// TwinCAT 3 PLC project Testing
// ProgramVersion: 3.1.4026.17
// libraries:
//   Tc2_Standard, * (Beckhoff Automation GmbH)
//   Tc2_System, * (Beckhoff Automation GmbH)
//   [TcForge], * (Home)
//   TcUnit, * (www.tcunit.org)
// project tree:
//   POUs/ MAIN.TcPOU, FB_DeviceBase_Probe.TcPOU, FB_DigitalInput_Probe.TcPOU, FB_TwoPosActuator_Probe.TcPOU, FB_AnalogInput_Probe.TcPOU, FB_AnalogOutput_Probe.TcPOU, FB_StateMachine_Probe.TcPOU
//   / Testing.TcTTO
//   Tests/ FB_F_ValidateRequester_Test.TcPOU, FB_BitMatrix64_Test.TcPOU, FB_Permissives_Test.TcPOU, FB_Interlock_Test.TcPOU, FB_AlarmSimple_Test.TcPOU, FB_AlarmLimit_Test.TcPOU, FB_DeviceBase_Test.TcPOU, FB_LPF_FirstOrder_IIR_Test.TcPOU, FB_DigitalOutput_Test.TcPOU, FB_DigitalInput_Test.TcPOU, FB_TwoPosActuator_Test.TcPOU, FB_AnalogInput_Test.TcPOU, FB_AnalogOutput_Test.TcPOU, FB_AlarmThreshold_Test.TcPOU, FB_AlarmDeviation_Test.TcPOU, FB_Step_Test.TcPOU, FB_StateMachine_Test.TcPOU
// (motion and I/O tree: see PLC project tcforge)
// real-time tasks:
//   TASK Testing: cycle T#10ms, priority 2, ADS port 351
//   TASK PlcTask: cycle T#10ms, priority 1, ADS port 350

CONFIGURATION Testing
    RESOURCE PLC ON TwinCAT3
        TASK Testing(INTERVAL := T#10ms, PRIORITY := 2);
        PROGRAM MAIN WITH Testing : MAIN;
    END_RESOURCE
END_CONFIGURATION

// ---- POUs/MAIN.TcPOU
PROGRAM MAIN
VAR
    fbValidateRequester_Test : FB_F_ValidateRequester_Test;
    fbBitMatrix64_Test       : FB_BitMatrix64_Test;
    fbPermissives_Test       : FB_Permissives_Test;
    fbInterlock_Test         : FB_Interlock_Test;
    fbAlarmSimple_Test       : FB_AlarmSimple_Test;
    fbAlarmLimit_Test        : FB_AlarmLimit_Test;
    fbDeviceBase_Test        : FB_DeviceBase_Test;
    fbLpfFirstOrder_Test     : FB_LPF_FirstOrder_IIR_Test;
    fbDigitalOutput_Test     : FB_DigitalOutput_Test;
    fbDigitalInput_Test      : FB_DigitalInput_Test;
    fbTwoPosActuator_Test    : FB_TwoPosActuator_Test;
    fbAnalogInput_Test       : FB_AnalogInput_Test;
    fbAnalogOutput_Test      : FB_AnalogOutput_Test;
    fbAlarmThreshold_Test    : FB_AlarmThreshold_Test;
    fbAlarmDeviation_Test    : FB_AlarmDeviation_Test;
    fbStep_Test              : FB_Step_Test;
    fbStateMachine_Test      : FB_StateMachine_Test;
END_VAR

TcUnit.RUN();

END_PROGRAM

// ---- Tests/FB_F_ValidateRequester_Test.TcPOU
FUNCTION_BLOCK FB_F_ValidateRequester_Test EXTENDS TcUnit.FB_TestSuite
VAR
END_VAR

AcceptsNormally();
AcceptsProgramWhenLocked();
RejectsOperatorWhenLocked();
RejectsWhenFaulted();

METHOD AcceptsNormally
VAR
    nExpected : DINT := TcForge.E_RpcMethodResponse.ACCEPTED;
    nActual   : DINT;
END_VAR
TEST('AcceptsNormally');

nActual := TcForge.F_ValidateRequester(
    eRequester    := TcForge.E_Requester.OPERATOR,
    bSourceLocked := FALSE,
    bFaulted      := FALSE);

AssertEquals_DINT(
    Expected := nExpected,
    Actual   := nActual,
    Message  := 'Should accept when there are no restrictions');

TEST_FINISHED();
END_METHOD

METHOD AcceptsProgramWhenLocked
VAR
    nExpected : DINT := TcForge.E_RpcMethodResponse.ACCEPTED;
    nActual   : DINT;
END_VAR
TEST('AcceptsProgramWhenLocked');

nActual := TcForge.F_ValidateRequester(
    eRequester    := TcForge.E_Requester.PROG,
    bSourceLocked := TRUE,
    bFaulted      := FALSE);

AssertEquals_DINT(
    Expected := nExpected,
    Actual   := nActual,
    Message  := 'PROG requester should be accepted even when source is locked');

TEST_FINISHED();
END_METHOD

METHOD RejectsOperatorWhenLocked
VAR
    nExpected : DINT := TcForge.E_RpcMethodResponse.REJECTED_SOURCE_NOT_ALLOWED;
    nActual   : DINT;
END_VAR
TEST('RejectsOperatorWhenLocked');

nActual := TcForge.F_ValidateRequester(
    eRequester    := TcForge.E_Requester.OPERATOR,
    bSourceLocked := TRUE,
    bFaulted      := FALSE);

AssertEquals_DINT(
    Expected := nExpected,
    Actual   := nActual,
    Message  := 'OPERATOR must be rejected when source is locked');

TEST_FINISHED();
END_METHOD

METHOD RejectsWhenFaulted
VAR
    nExpected : DINT := TcForge.E_RpcMethodResponse.REJECTED_FAULTED;
    nActual   : DINT;
END_VAR
TEST('RejectsWhenFaulted');

nActual := TcForge.F_ValidateRequester(
    eRequester    := TcForge.E_Requester.OPERATOR,
    bSourceLocked := FALSE,
    bFaulted      := TRUE);

AssertEquals_DINT(
    Expected := nExpected,
    Actual   := nActual,
    Message  := 'Should reject when faulted');

TEST_FINISHED();
END_METHOD

END_FUNCTION_BLOCK

// ---- Tests/FB_BitMatrix64_Test.TcPOU
// Unit tests for FB_BitMatrix64 — the shared 64-bit condition-matrix core
// consumed by FB_Permissives (non-latching) and FB_Interlock (latching).
// Covers the behaviours both composers rely on: live bit semantics, active-
// mask tracking, mapping timeout, "just unmapped while bad" events, first-
// failure ordering, bypass accept/reject rules, and clear operations.
//
// Each test owns a fresh FB_BitMatrix64 instance via METHOD-local VARs so
// cycle counters and internal state do not leak between tests.
FUNCTION_BLOCK FB_BitMatrix64_Test EXTENDS TcUnit.FB_TestSuite

InitialStateAllGood();
MapInputMarksActiveAndValue();
MapInputBadValueClearsLiveBit();
MapInputOutOfRangeIsNoOp();
MappingTimeoutUnmapsAndRestoresGood();
JustUnmappedBadFiresWhenBadAtUnmap();
JustUnmappedBadSilentWhenGoodAtUnmap();
FirstFailureRecordsFirstBadBit();
SetBypassAcceptsWhenBypassable();
SetBypassRejectsWhenNotBypassable();
SetBypassClearAlwaysAllowed();
SetBypassInvalidBitIndex();
ClearBypassClearsAll();
ClearFirstFailureResets();

METHOD InitialStateAllGood
VAR
    fb : TcForge.FB_BitMatrix64;
END_VAR
TEST('InitialStateAllGood');

// Before any body call, default initialisers should mark every bit good
// and no bit active / bypassed / tripped.
AssertEquals_ULINT(
    Expected := 16#FFFFFFFFFFFFFFFF,
    Actual   := fb.nLiveBits,
    Message  := 'Fresh instance: nLiveBits should be all-good');
AssertEquals_ULINT(
    Expected := 0,
    Actual   := fb.nActiveMask,
    Message  := 'Fresh instance: nActiveMask should be empty');
AssertEquals_ULINT(
    Expected := 0,
    Actual   := fb.nBypassMask,
    Message  := 'Fresh instance: nBypassMask should be empty');
AssertEquals_UDINT(
    Expected := 999,
    Actual   := fb.nFirstFailureBitIndex,
    Message  := 'Fresh instance: nFirstFailureBitIndex should be sentinel 999');
AssertEquals_ULINT(
    Expected := 0,
    Actual   := fb.nJustUnmappedBad,
    Message  := 'Fresh instance: nJustUnmappedBad should be empty');

TEST_FINISHED();
END_METHOD

METHOD MapInputMarksActiveAndValue
VAR
    fb      : TcForge.FB_BitMatrix64;
    bitMask : ULINT;
END_VAR
TEST('MapInputMarksActiveAndValue');

bitMask := SHL(ULINT#1, 5);

fb.MapInput(bitIndex := 5, inputValue := TRUE);
fb();

AssertTrue(
    Condition := (fb.nActiveMask AND bitMask) <> 0,
    Message   := 'Bit 5 should be in nActiveMask after MapInput(5, TRUE)');
AssertTrue(
    Condition := (fb.nLiveBits AND bitMask) <> 0,
    Message   := 'Bit 5 should be good (1) in nLiveBits after MapInput(5, TRUE)');

TEST_FINISHED();
END_METHOD

METHOD MapInputBadValueClearsLiveBit
VAR
    fb      : TcForge.FB_BitMatrix64;
    bitMask : ULINT;
END_VAR
TEST('MapInputBadValueClearsLiveBit');

bitMask := SHL(ULINT#1, 5);

fb.MapInput(bitIndex := 5, inputValue := FALSE);
fb();

AssertTrue(
    Condition := (fb.nActiveMask AND bitMask) <> 0,
    Message   := 'Bit 5 should still be active even when value is FALSE');
AssertTrue(
    Condition := (fb.nLiveBits AND bitMask) = 0,
    Message   := 'Bit 5 should be bad (0) in nLiveBits after MapInput(5, FALSE)');

TEST_FINISHED();
END_METHOD

METHOD MapInputOutOfRangeIsNoOp
VAR
    fb : TcForge.FB_BitMatrix64;
END_VAR
TEST('MapInputOutOfRangeIsNoOp');

// Bit 64 is outside the 0..63 range; MapInput must silently reject it.
fb.MapInput(bitIndex := 64, inputValue := FALSE);
fb();

AssertEquals_ULINT(
    Expected := 0,
    Actual   := fb.nActiveMask,
    Message  := 'MapInput with bitIndex > 63 must not touch nActiveMask');
AssertEquals_ULINT(
    Expected := 16#FFFFFFFFFFFFFFFF,
    Actual   := fb.nLiveBits,
    Message  := 'MapInput with bitIndex > 63 must not touch nLiveBits');

TEST_FINISHED();
END_METHOD

METHOD MappingTimeoutUnmapsAndRestoresGood
VAR
    fb      : TcForge.FB_BitMatrix64;
    bitMask : ULINT;
    i       : UDINT;
END_VAR
TEST('MappingTimeoutUnmapsAndRestoresGood');

bitMask := SHL(ULINT#1, 5);

// Map bit 5 once as bad, then stop feeding. After MAPPING_TIMEOUT (=10)
// unreferenced cycles the bit must be unmapped and snap back to good.
fb.MapInput(bitIndex := 5, inputValue := FALSE);
fb();  // cycle 1 — freshly mapped

FOR i := 1 TO 12 DO  // run past the 10-cycle timeout
    fb();
END_FOR;

AssertTrue(
    Condition := (fb.nActiveMask AND bitMask) = 0,
    Message   := 'Bit 5 should be unmapped after MAPPING_TIMEOUT cycles without refresh');
AssertTrue(
    Condition := (fb.nLiveBits AND bitMask) <> 0,
    Message   := 'Bit 5 should snap back to good once unmapped');

TEST_FINISHED();
END_METHOD

METHOD JustUnmappedBadFiresWhenBadAtUnmap
VAR
    fb        : TcForge.FB_BitMatrix64;
    bitMask   : ULINT;
    i         : UDINT;
    sawEvent  : BOOL;
END_VAR
TEST('JustUnmappedBadFiresWhenBadAtUnmap');

bitMask := SHL(ULINT#1, 5);

// Map bit 5 as BAD, then stop feeding. Somewhere in the next cycles the
// cleanup loop will unmap it; that tick must publish the event via
// nJustUnmappedBad so latching callers (FB_Interlock) can remember it.
fb.MapInput(bitIndex := 5, inputValue := FALSE);
fb();

sawEvent := FALSE;
FOR i := 1 TO 15 DO
    fb();
    IF (fb.nJustUnmappedBad AND bitMask) <> 0 THEN
        sawEvent := TRUE;
    END_IF;
END_FOR;

AssertTrue(
    Condition := sawEvent,
    Message   := 'nJustUnmappedBad should fire for bit 5 during the timeout-unmap cycle');

// Event must be edge-style: once the unmap cycle passes, subsequent cycles
// reset the output.
AssertEquals_ULINT(
    Expected := 0,
    Actual   := fb.nJustUnmappedBad,
    Message  := 'nJustUnmappedBad should clear on cycles after the unmap event');

TEST_FINISHED();
END_METHOD

METHOD JustUnmappedBadSilentWhenGoodAtUnmap
VAR
    fb       : TcForge.FB_BitMatrix64;
    bitMask  : ULINT;
    i        : UDINT;
    sawEvent : BOOL;
END_VAR
TEST('JustUnmappedBadSilentWhenGoodAtUnmap');

bitMask := SHL(ULINT#1, 5);

// Map bit 5 as GOOD then stop feeding. The timeout unmap still happens,
// but there is no "bad at unmap" memory to expose — event must stay clear.
fb.MapInput(bitIndex := 5, inputValue := TRUE);
fb();

sawEvent := FALSE;
FOR i := 1 TO 15 DO
    fb();
    IF (fb.nJustUnmappedBad AND bitMask) <> 0 THEN
        sawEvent := TRUE;
    END_IF;
END_FOR;

AssertFalse(
    Condition := sawEvent,
    Message   := 'nJustUnmappedBad must NOT fire when the bit was good at unmap');

TEST_FINISHED();
END_METHOD

METHOD FirstFailureRecordsFirstBadBit
VAR
    fb : TcForge.FB_BitMatrix64;
END_VAR
TEST('FirstFailureRecordsFirstBadBit');

// Cycle 1: bits 3 and 7 both mapped good; baseline is all good.
fb.MapInput(bitIndex := 3, inputValue := TRUE);
fb.MapInput(bitIndex := 7, inputValue := TRUE);
fb();

// Cycle 2: both drop to bad in the same scan. The body scans bits 0..63 in
// order, so the lower-index bit (3) wins the first-failure slot.
fb.MapInput(bitIndex := 3, inputValue := FALSE);
fb.MapInput(bitIndex := 7, inputValue := FALSE);
fb();

AssertEquals_UDINT(
    Expected := 3,
    Actual   := fb.nFirstFailureBitIndex,
    Message  := 'First-failure index should be the lowest-numbered bit that went bad');

TEST_FINISHED();
END_METHOD

METHOD SetBypassAcceptsWhenBypassable
VAR
    fb       : TcForge.FB_BitMatrix64;
    bitMask  : ULINT;
    response : TcForge.E_RpcMethodResponse;
END_VAR
TEST('SetBypassAcceptsWhenBypassable');

bitMask := SHL(ULINT#1, 3);

response := fb.SetBypass(
    bitIndex        := 3,
    bEnable         := TRUE,
    nBypassableMask := bitMask);

AssertEquals_DINT(
    Expected := TcForge.E_RpcMethodResponse.ACCEPTED,
    Actual   := response,
    Message  := 'SetBypass should accept when the bit is configured as bypassable');
AssertTrue(
    Condition := (fb.nBypassMask AND bitMask) <> 0,
    Message   := 'nBypassMask should reflect the accepted bypass');

TEST_FINISHED();
END_METHOD

METHOD SetBypassRejectsWhenNotBypassable
VAR
    fb       : TcForge.FB_BitMatrix64;
    response : TcForge.E_RpcMethodResponse;
END_VAR
TEST('SetBypassRejectsWhenNotBypassable');

// Caller supplies an empty bypassable mask, so any enable attempt must be
// rejected regardless of which bit is targeted.
response := fb.SetBypass(
    bitIndex        := 3,
    bEnable         := TRUE,
    nBypassableMask := 0);

AssertEquals_DINT(
    Expected := TcForge.E_RpcMethodResponse.REJECTED_BYPASS_NOT_ALLOWED,
    Actual   := response,
    Message  := 'SetBypass must reject enable when the bit is not configured as bypassable');
AssertEquals_ULINT(
    Expected := 0,
    Actual   := fb.nBypassMask,
    Message  := 'nBypassMask must stay empty after a rejected SetBypass');

TEST_FINISHED();
END_METHOD

METHOD SetBypassClearAlwaysAllowed
VAR
    fb       : TcForge.FB_BitMatrix64;
    response : TcForge.E_RpcMethodResponse;
END_VAR
TEST('SetBypassClearAlwaysAllowed');

// Clearing a bypass is always safe: even if the bit is not configured as
// bypassable, removing a bypass cannot violate any safety invariant.
response := fb.SetBypass(
    bitIndex        := 3,
    bEnable         := FALSE,
    nBypassableMask := 0);

AssertEquals_DINT(
    Expected := TcForge.E_RpcMethodResponse.ACCEPTED,
    Actual   := response,
    Message  := 'Clearing a bypass must always be accepted');

TEST_FINISHED();
END_METHOD

METHOD SetBypassInvalidBitIndex
VAR
    fb       : TcForge.FB_BitMatrix64;
    response : TcForge.E_RpcMethodResponse;
END_VAR
TEST('SetBypassInvalidBitIndex');

response := fb.SetBypass(
    bitIndex        := 64,
    bEnable         := TRUE,
    nBypassableMask := 16#FFFFFFFFFFFFFFFF);

AssertEquals_DINT(
    Expected := TcForge.E_RpcMethodResponse.REJECTED_INVALID_PARAMETER,
    Actual   := response,
    Message  := 'SetBypass must reject bitIndex > 63 with REJECTED_INVALID_PARAMETER');

TEST_FINISHED();
END_METHOD

METHOD ClearBypassClearsAll
VAR
    fb : TcForge.FB_BitMatrix64;
END_VAR
TEST('ClearBypassClearsAll');

// Bypass two separate bits, then clear them in one call.
fb.SetBypass(bitIndex := 2, bEnable := TRUE, nBypassableMask := 16#FFFFFFFFFFFFFFFF);
fb.SetBypass(bitIndex := 9, bEnable := TRUE, nBypassableMask := 16#FFFFFFFFFFFFFFFF);
fb.ClearBypass();

AssertEquals_ULINT(
    Expected := 0,
    Actual   := fb.nBypassMask,
    Message  := 'ClearBypass must wipe nBypassMask in a single call');

TEST_FINISHED();
END_METHOD

METHOD ClearFirstFailureResets
VAR
    fb : TcForge.FB_BitMatrix64;
END_VAR
TEST('ClearFirstFailureResets');

// Produce a real first-failure sequence, then clear it.
fb.MapInput(bitIndex := 3, inputValue := TRUE);
fb();
fb.MapInput(bitIndex := 3, inputValue := FALSE);
fb();

AssertEquals_UDINT(
    Expected := 3,
    Actual   := fb.nFirstFailureBitIndex,
    Message  := 'Precondition: failure sequence should record bit 3');

fb.ClearFirstFailure();

AssertEquals_UDINT(
    Expected := 999,
    Actual   := fb.nFirstFailureBitIndex,
    Message  := 'ClearFirstFailure must restore the sentinel 999');

TEST_FINISHED();
END_METHOD

END_FUNCTION_BLOCK

// ---- Tests/FB_Permissives_Test.TcPOU
// Integration tests for FB_Permissives on top of FB_BitMatrix64.
// FB_BitMatrix64_Test already covers the shared matrix mechanics, so this
// suite focuses on permissive-specific behaviour:
//   - non-latching rollup: sts.bOK tracks live inputs in both directions
//   - bypass forces the bit good in the rollup
//   - Reset() clears bypass (the only thing Reset needs to do here — the
//     permissive has no latched state to snap)
//   - cfg.nBypassable gating propagates through SetBypass
//   - first-failure and faceplate surfaces reflect core state
FUNCTION_BLOCK FB_Permissives_Test EXTENDS TcUnit.FB_TestSuite

InitialStateOk();
BadMappedBitFailsOK();
RecoveryFlipsOKTrueAgain();
BypassForcesGoodInRollup();
ResetClearsBypass();
SetBypassRejectsWhenNotBypassable();
FirstFailureIndexPropagates();
FaceplateReflectsLiveState();

METHOD InitialStateOk
VAR
    fb : TcForge.FB_Permissives;
END_VAR
TEST('InitialStateOk');

fb();  // no MapInput calls — unmapped bits default good

AssertTrue(
    Condition := fb.sts.bOK,
    Message   := 'Fresh permissives with no mappings should report bOK = TRUE');
AssertEquals_ULINT(
    Expected := 16#FFFFFFFFFFFFFFFF,
    Actual   := fb.sts.nPermissives,
    Message  := 'Fresh permissives rollup should be all-good');
AssertEquals_UDINT(
    Expected := 999,
    Actual   := fb.sts.nFirstFailureBitIndex,
    Message  := 'Fresh permissives should expose the sentinel first-failure index');

TEST_FINISHED();
END_METHOD

METHOD BadMappedBitFailsOK
VAR
    fb      : TcForge.FB_Permissives;
    bitMask : ULINT;
END_VAR
TEST('BadMappedBitFailsOK');

bitMask := SHL(ULINT#1, 5);

fb.MapInput(bitIndex := 5, inputValue := FALSE);
fb();

AssertFalse(
    Condition := fb.sts.bOK,
    Message   := 'bOK must be FALSE when any mapped bit is bad');
AssertTrue(
    Condition := (fb.sts.nPermissives AND bitMask) = 0,
    Message   := 'Bit 5 should show as bad in the rollup');

TEST_FINISHED();
END_METHOD

METHOD RecoveryFlipsOKTrueAgain
VAR
    fb : TcForge.FB_Permissives;
END_VAR
TEST('RecoveryFlipsOKTrueAgain');

// This is the defining permissive behaviour: when the condition recovers,
// bOK returns to TRUE on the *same* cycle, with no Reset() required.
fb.MapInput(bitIndex := 5, inputValue := FALSE);
fb();

AssertFalse(
    Condition := fb.sts.bOK,
    Message   := 'Precondition: bOK should be FALSE while bit 5 is bad');

fb.MapInput(bitIndex := 5, inputValue := TRUE);
fb();

AssertTrue(
    Condition := fb.sts.bOK,
    Message   := 'Permissive is non-latching: bOK must flip back to TRUE the cycle the input recovers');

TEST_FINISHED();
END_METHOD

METHOD BypassForcesGoodInRollup
VAR
    fb       : TcForge.FB_Permissives;
    bitMask  : ULINT;
    response : TcForge.E_RpcMethodResponse;
END_VAR
TEST('BypassForcesGoodInRollup');

bitMask := SHL(ULINT#1, 5);
fb.cfg.nBypassable := bitMask;

fb.MapInput(bitIndex := 5, inputValue := FALSE);
response := fb.SetBypass(bitIndex := 5, bEnable := TRUE);
fb();

AssertEquals_DINT(
    Expected := TcForge.E_RpcMethodResponse.ACCEPTED,
    Actual   := response,
    Message  := 'SetBypass should accept when the bit is flagged bypassable in cfg');
AssertTrue(
    Condition := fb.sts.bOK,
    Message   := 'A bypassed bit must be forced good in the rollup');
AssertTrue(
    Condition := (fb.sts.nBypassMask AND bitMask) <> 0,
    Message   := 'sts.nBypassMask should surface the active bypass');

TEST_FINISHED();
END_METHOD

METHOD ResetClearsBypass
VAR
    fb      : TcForge.FB_Permissives;
    bitMask : ULINT;
END_VAR
TEST('ResetClearsBypass');

bitMask := SHL(ULINT#1, 3);
fb.cfg.nBypassable := bitMask;

fb.SetBypass(bitIndex := 3, bEnable := TRUE);
fb();

AssertTrue(
    Condition := (fb.sts.nBypassMask AND bitMask) <> 0,
    Message   := 'Precondition: bit 3 bypass should be active before Reset()');

fb.Reset();
fb();

AssertEquals_ULINT(
    Expected := 0,
    Actual   := fb.sts.nBypassMask,
    Message  := 'Reset() on a permissive must clear every bypass bit');

TEST_FINISHED();
END_METHOD

METHOD SetBypassRejectsWhenNotBypassable
VAR
    fb       : TcForge.FB_Permissives;
    response : TcForge.E_RpcMethodResponse;
END_VAR
TEST('SetBypassRejectsWhenNotBypassable');

fb.cfg.nBypassable := 0;

response := fb.SetBypass(bitIndex := 5, bEnable := TRUE);
fb();

AssertEquals_DINT(
    Expected := TcForge.E_RpcMethodResponse.REJECTED_BYPASS_NOT_ALLOWED,
    Actual   := response,
    Message  := 'SetBypass must honour cfg.nBypassable and reject non-allowed bits');
AssertEquals_ULINT(
    Expected := 0,
    Actual   := fb.sts.nBypassMask,
    Message  := 'A rejected bypass must leave nBypassMask untouched');

TEST_FINISHED();
END_METHOD

METHOD FirstFailureIndexPropagates
VAR
    fb : TcForge.FB_Permissives;
END_VAR
TEST('FirstFailureIndexPropagates');

fb.MapInput(bitIndex := 7, inputValue := TRUE);
fb();

fb.MapInput(bitIndex := 7, inputValue := FALSE);
fb();

AssertEquals_UDINT(
    Expected := 7,
    Actual   := fb.sts.nFirstFailureBitIndex,
    Message  := 'sts.nFirstFailureBitIndex should surface the core first-failure index');

TEST_FINISHED();
END_METHOD

METHOD FaceplateReflectsLiveState
VAR
    fb : TcForge.FB_Permissives;
END_VAR
TEST('FaceplateReflectsLiveState');

fb.cfg.nBypassable   := SHL(ULINT#1, 4);
fb.cfg.aNames[4]     := 'TestPerm';

fb.MapInput(bitIndex := 4, inputValue := FALSE);
fb();

AssertEquals_STRING(
    Expected := 'TestPerm',
    Actual   := fb.sts.aFaceplates[4].name,
    Message  := 'Faceplate should mirror cfg.aNames[i]');
AssertFalse(
    Condition := fb.sts.aFaceplates[4].ok,
    Message   := 'Faceplate ok should mirror the rollup for that bit');
AssertTrue(
    Condition := fb.sts.aFaceplates[4].mapped,
    Message   := 'Faceplate mapped should mirror nActiveMask for that bit');
AssertTrue(
    Condition := fb.sts.aFaceplates[4].bypassable,
    Message   := 'Faceplate bypassable should mirror cfg.nBypassable for that bit');

TEST_FINISHED();
END_METHOD

END_FUNCTION_BLOCK

// ---- Tests/FB_Interlock_Test.TcPOU
// Integration tests for FB_Interlock on top of FB_BitMatrix64.
// FB_BitMatrix64_Test already covers the shared matrix mechanics, so this
// suite focuses on interlock-specific behaviour:
//   - once a mapped bit goes bad it stays bad (latching), even if the
//     underlying signal recovers on its own
//   - Reset() snaps the latch to the current live value; a still-bad bit
//     stays bad (reset is not a safety override)
//   - unmapped-bad memory keeps bOK FALSE after a bit becomes unmapped
//     while it was bad, and survives until Reset() clears it
//   - bypass still forces a bit good in the effective rollup
//   - Reset() intentionally preserves bypass state
FUNCTION_BLOCK FB_Interlock_Test EXTENDS TcUnit.FB_TestSuite

InitialStateOk();
BadMappedBitLatches();
RecoveryDoesNotClearLatch();
ResetClearsLatchAfterRecovery();
ResetWithActiveBadLeavesItBad();
UnmappedBadMemoryKeepsBOkFalse();
ResetClearsUnmappedBadMemory();
BypassForcesGoodInRollup();
ResetPreservesBypass();

METHOD InitialStateOk
VAR
    fb : TcForge.FB_Interlock;
END_VAR
TEST('InitialStateOk');

fb();

AssertTrue(
    Condition := fb.sts.bOK,
    Message   := 'Fresh interlock with no mappings should report bOK = TRUE');
AssertEquals_ULINT(
    Expected := 16#FFFFFFFFFFFFFFFF,
    Actual   := fb.sts.nInterlocks,
    Message  := 'Fresh interlock rollup should be all-good');
AssertEquals_UDINT(
    Expected := 999,
    Actual   := fb.sts.nFirstFailureBitIndex,
    Message  := 'Fresh interlock should expose the sentinel first-failure index');

TEST_FINISHED();
END_METHOD

METHOD BadMappedBitLatches
VAR
    fb      : TcForge.FB_Interlock;
    bitMask : ULINT;
END_VAR
TEST('BadMappedBitLatches');

bitMask := SHL(ULINT#1, 5);

fb.MapInput(bitIndex := 5, inputValue := FALSE);
fb();

AssertFalse(
    Condition := fb.sts.bOK,
    Message   := 'bOK must be FALSE while bit 5 is bad');
AssertTrue(
    Condition := (fb.sts.nInterlocks AND bitMask) = 0,
    Message   := 'Bit 5 should show as bad in the effective rollup');

TEST_FINISHED();
END_METHOD

METHOD RecoveryDoesNotClearLatch
VAR
    fb : TcForge.FB_Interlock;
END_VAR
TEST('RecoveryDoesNotClearLatch');

// This is the defining interlock behaviour: once bad, stays bad until
// Reset() is explicitly called, even after the input recovers on its own.
fb.MapInput(bitIndex := 5, inputValue := FALSE);
fb();

AssertFalse(
    Condition := fb.sts.bOK,
    Message   := 'Precondition: bOK should be FALSE while bit 5 is bad');

fb.MapInput(bitIndex := 5, inputValue := TRUE);
fb();
fb.MapInput(bitIndex := 5, inputValue := TRUE);
fb();

AssertFalse(
    Condition := fb.sts.bOK,
    Message   := 'Interlock must stay latched FALSE after the input recovers until Reset() is called');

TEST_FINISHED();
END_METHOD

METHOD ResetClearsLatchAfterRecovery
VAR
    fb : TcForge.FB_Interlock;
END_VAR
TEST('ResetClearsLatchAfterRecovery');

// Fault -> recover -> Reset() -> bOK TRUE.
fb.MapInput(bitIndex := 5, inputValue := FALSE);
fb();
fb.MapInput(bitIndex := 5, inputValue := TRUE);
fb();

fb.Reset();
fb.MapInput(bitIndex := 5, inputValue := TRUE);
fb();

AssertTrue(
    Condition := fb.sts.bOK,
    Message   := 'Reset() after recovery must clear the latch and restore bOK = TRUE');

TEST_FINISHED();
END_METHOD

METHOD ResetWithActiveBadLeavesItBad
VAR
    fb : TcForge.FB_Interlock;
END_VAR
TEST('ResetWithActiveBadLeavesItBad');

// Reset() is a latch clear, not a safety override. If the live condition
// is still bad when Reset() is called, bOK must stay FALSE.
fb.MapInput(bitIndex := 5, inputValue := FALSE);
fb();

fb.Reset();
fb.MapInput(bitIndex := 5, inputValue := FALSE);
fb();

AssertFalse(
    Condition := fb.sts.bOK,
    Message   := 'Reset() while the condition is still bad must NOT clear the failure');

TEST_FINISHED();
END_METHOD

METHOD UnmappedBadMemoryKeepsBOkFalse
VAR
    fb : TcForge.FB_Interlock;
    i  : UDINT;
END_VAR
TEST('UnmappedBadMemoryKeepsBOkFalse');

// Map bit 5 as bad exactly once, then stop feeding. After MAPPING_TIMEOUT
// the bit is removed from the active mask — but the interlock must
// remember it was bad at the moment of unmap and keep bOK FALSE until
// Reset() is called. This is the key safety invariant that survived the
// FB_BitMatrix64 extraction.
fb.MapInput(bitIndex := 5, inputValue := FALSE);
fb();

FOR i := 1 TO 15 DO
    fb();
END_FOR;

AssertFalse(
    Condition := fb.sts.bOK,
    Message   := 'Interlock must stay FALSE after a bit became unmapped while bad');

TEST_FINISHED();
END_METHOD

METHOD ResetClearsUnmappedBadMemory
VAR
    fb : TcForge.FB_Interlock;
    i  : UDINT;
END_VAR
TEST('ResetClearsUnmappedBadMemory');

fb.MapInput(bitIndex := 5, inputValue := FALSE);
fb();
FOR i := 1 TO 15 DO
    fb();
END_FOR;

AssertFalse(
    Condition := fb.sts.bOK,
    Message   := 'Precondition: unmapped-bad memory should be holding bOK FALSE');

fb.Reset();
fb();

AssertTrue(
    Condition := fb.sts.bOK,
    Message   := 'Reset() must clear the unmapped-bad memory and restore bOK = TRUE');

TEST_FINISHED();
END_METHOD

METHOD BypassForcesGoodInRollup
VAR
    fb       : TcForge.FB_Interlock;
    bitMask  : ULINT;
    response : TcForge.E_RpcMethodResponse;
END_VAR
TEST('BypassForcesGoodInRollup');

bitMask := SHL(ULINT#1, 5);
fb.cfg.nBypassable := bitMask;

fb.MapInput(bitIndex := 5, inputValue := FALSE);
response := fb.SetBypass(bitIndex := 5, bEnable := TRUE);
fb();

AssertEquals_DINT(
    Expected := TcForge.E_RpcMethodResponse.ACCEPTED,
    Actual   := response,
    Message  := 'SetBypass should accept when the bit is flagged bypassable in cfg');
AssertTrue(
    Condition := fb.sts.bOK,
    Message   := 'A bypassed bit must be forced good in the effective rollup');

TEST_FINISHED();
END_METHOD

METHOD ResetPreservesBypass
VAR
    fb      : TcForge.FB_Interlock;
    bitMask : ULINT;
END_VAR
TEST('ResetPreservesBypass');

bitMask := SHL(ULINT#1, 5);
fb.cfg.nBypassable := bitMask;

fb.SetBypass(bitIndex := 5, bEnable := TRUE);
fb();

AssertTrue(
    Condition := (fb.sts.nBypassMask AND bitMask) <> 0,
    Message   := 'Precondition: bit 5 bypass should be active before Reset()');

fb.Reset();
fb();

AssertTrue(
    Condition := (fb.sts.nBypassMask AND bitMask) <> 0,
    Message   := 'Reset() on an interlock must PRESERVE bypass state (per the public contract)');

TEST_FINISHED();
END_METHOD

END_FUNCTION_BLOCK

// ---- Tests/FB_AlarmSimple_Test.TcPOU
// FB_AlarmSimple is the thinnest concrete child of FB_AlarmBase, so this
// suite doubles as the test harness for the shared alarm contract:
// enable gating, raw -> active rollup, latch + ack state machine, severity
// propagation, message echo, source-lock gating on Ack().
//
// Debounce (TON/TOF) is intentionally exercised with T#0MS delays; the
// debounce primitive itself is IEC standard and testing its timing under
// TcUnit is awkward because a suite body runs once per task cycle. Every
// test below therefore lets tOnDelay / tOffDelay stay at zero and focuses
// on the alarm logic that sits on top of the debounced signal.
FUNCTION_BLOCK FB_AlarmSimple_Test EXTENDS TcUnit.FB_TestSuite

DisabledSuppressesEverything();
SelfClearingTracksInput();
LatchingHoldsAfterClearWithoutAck();
AckAfterClearReleasesLatch();
AckWhileActiveFlipsAckedButNotLatch();
SeverityFollowsActiveState();
MessageEchoedFromCfg();
DisableClearsActiveLatch();
LockedSourceRejectsOperatorAck();
AckWithNoLatchIsNoOp();

METHOD DisabledSuppressesEverything
VAR
    fb : TcForge.FB_AlarmSimple;
END_VAR
TEST('DisabledSuppressesEverything');

// cfg.bEnable defaults to FALSE; even with the input firing, the alarm
// must stay inert and report severity NONE.
fb.cfg.common.eSeverity := TcForge.E_AlarmSeverity.CRITICAL;

fb(inpActive := TRUE);

AssertFalse(
    Condition := fb.sts.active,
    Message   := 'Disabled alarm must not go active');
AssertEquals_USINT(
    Expected := TcForge.E_AlarmSeverity.NONE,
    Actual   := fb.sts.eSeverity,
    Message  := 'Disabled alarm must report severity NONE');

TEST_FINISHED();
END_METHOD

METHOD SelfClearingTracksInput
VAR
    fb : TcForge.FB_AlarmSimple;
END_VAR
TEST('SelfClearingTracksInput');

// bRequireAck = FALSE => no latch. active follows the debounced input
// in both directions.
fb.cfg.common.bEnable     := TRUE;
fb.cfg.common.bRequireAck := FALSE;
fb.cfg.common.eSeverity   := TcForge.E_AlarmSeverity.WARNING;

fb(inpActive := TRUE);
AssertTrue(
    Condition := fb.sts.active,
    Message   := 'Non-latching alarm should go active when the input is TRUE');

fb(inpActive := FALSE);
AssertFalse(
    Condition := fb.sts.active,
    Message   := 'Non-latching alarm should clear the same cycle the input clears');
AssertFalse(
    Condition := fb.sts.latched,
    Message   := 'Non-latching alarm must never expose latched');

TEST_FINISHED();
END_METHOD

METHOD LatchingHoldsAfterClearWithoutAck
VAR
    fb : TcForge.FB_AlarmSimple;
END_VAR
TEST('LatchingHoldsAfterClearWithoutAck');

fb.cfg.common.bEnable     := TRUE;
fb.cfg.common.bRequireAck := TRUE;
fb.cfg.common.eSeverity   := TcForge.E_AlarmSeverity.CRITICAL;

fb(inpActive := TRUE);
AssertTrue(
    Condition := fb.sts.active,
    Message   := 'Latching alarm should go active when the input fires');
AssertTrue(
    Condition := fb.sts.latched,
    Message   := 'latched should indicate an un-acked latch');

fb(inpActive := FALSE);
AssertTrue(
    Condition := fb.sts.active,
    Message   := 'Latching alarm must stay active after the input clears until Ack()');

TEST_FINISHED();
END_METHOD

METHOD AckAfterClearReleasesLatch
VAR
    fb       : TcForge.FB_AlarmSimple;
    response : TcForge.E_RpcMethodResponse;
END_VAR
TEST('AckAfterClearReleasesLatch');

fb.cfg.common.bEnable     := TRUE;
fb.cfg.common.bRequireAck := TRUE;
fb.cfg.common.eSeverity   := TcForge.E_AlarmSeverity.WARNING;

// Trip, clear the condition, then ack — latch should release next cycle.
fb(inpActive := TRUE);
fb(inpActive := FALSE);

response := fb.Ack(eRequester := TcForge.E_Requester.OPERATOR);
fb(inpActive := FALSE);

AssertEquals_DINT(
    Expected := TcForge.E_RpcMethodResponse.ACCEPTED,
    Actual   := response,
    Message  := 'Ack() with no source lock should be accepted');
AssertFalse(
    Condition := fb.sts.active,
    Message   := 'Latch must release once condition has cleared AND Ack() has been called');

TEST_FINISHED();
END_METHOD

METHOD AckWhileActiveFlipsAckedButNotLatch
VAR
    fb : TcForge.FB_AlarmSimple;
END_VAR
TEST('AckWhileActiveFlipsAckedButNotLatch');

fb.cfg.common.bEnable     := TRUE;
fb.cfg.common.bRequireAck := TRUE;
fb.cfg.common.eSeverity   := TcForge.E_AlarmSeverity.CRITICAL;

// Condition still firing when the operator acks — valid middle state:
// active stays TRUE, acked becomes TRUE, latched becomes FALSE
// (operator has seen it but the process is still in the bad state).
fb(inpActive := TRUE);
fb.Ack(eRequester := TcForge.E_Requester.OPERATOR);
fb(inpActive := TRUE);

AssertTrue(
    Condition := fb.sts.active,
    Message   := 'active should remain TRUE while the condition is still firing');
AssertTrue(
    Condition := fb.sts.acked,
    Message   := 'acked should be TRUE after an accepted Ack()');
AssertFalse(
    Condition := fb.sts.latched,
    Message   := 'latched should drop once the latch has been acknowledged');

TEST_FINISHED();
END_METHOD

METHOD SeverityFollowsActiveState
VAR
    fb : TcForge.FB_AlarmSimple;
END_VAR
TEST('SeverityFollowsActiveState');

fb.cfg.common.bEnable     := TRUE;
fb.cfg.common.bRequireAck := FALSE;
fb.cfg.common.eSeverity   := TcForge.E_AlarmSeverity.CRITICAL;

fb(inpActive := TRUE);
AssertEquals_USINT(
    Expected := TcForge.E_AlarmSeverity.CRITICAL,
    Actual   := fb.sts.eSeverity,
    Message  := 'Active alarm must publish the configured severity');

fb(inpActive := FALSE);
AssertEquals_USINT(
    Expected := TcForge.E_AlarmSeverity.NONE,
    Actual   := fb.sts.eSeverity,
    Message  := 'Inactive alarm must publish severity NONE (aggregators MAX() across alarms)');

TEST_FINISHED();
END_METHOD

METHOD MessageEchoedFromCfg
VAR
    fb : TcForge.FB_AlarmSimple;
END_VAR
TEST('MessageEchoedFromCfg');

fb.cfg.common.bEnable  := TRUE;
fb.cfg.common.sMessage := 'Cell door open';

fb(inpActive := FALSE);

AssertEquals_STRING(
    Expected := 'Cell door open',
    Actual   := fb.sts.sMessage,
    Message  := 'sts.sMessage must echo cfg.common.sMessage');

TEST_FINISHED();
END_METHOD

METHOD DisableClearsActiveLatch
VAR
    fb : TcForge.FB_AlarmSimple;
END_VAR
TEST('DisableClearsActiveLatch');

fb.cfg.common.bEnable     := TRUE;
fb.cfg.common.bRequireAck := TRUE;
fb.cfg.common.eSeverity   := TcForge.E_AlarmSeverity.CRITICAL;

// Latch, then disable. Flipping bEnable FALSE must force the alarm inert
// immediately — operator disables dominate any held latch.
fb(inpActive := TRUE);
AssertTrue(
    Condition := fb.sts.active,
    Message   := 'Precondition: latch should be active before disable');

fb.cfg.common.bEnable := FALSE;
fb(inpActive := TRUE);

AssertFalse(
    Condition := fb.sts.active,
    Message   := 'Disable must drop active even while the input is still firing');
AssertFalse(
    Condition := fb.sts.latched,
    Message   := 'Disable must clear latched');
AssertEquals_USINT(
    Expected := TcForge.E_AlarmSeverity.NONE,
    Actual   := fb.sts.eSeverity,
    Message  := 'Disable must drop severity back to NONE');

TEST_FINISHED();
END_METHOD

METHOD LockedSourceRejectsOperatorAck
VAR
    fb        : TcForge.FB_AlarmSimple;
    opResp    : TcForge.E_RpcMethodResponse;
    progResp  : TcForge.E_RpcMethodResponse;
END_VAR
TEST('LockedSourceRejectsOperatorAck');

fb.cfg.common.bEnable     := TRUE;
fb.cfg.common.bRequireAck := TRUE;
fb.cfg.common.eSeverity   := TcForge.E_AlarmSeverity.CRITICAL;

fb.LockSource(bLock := TRUE);
fb(inpActive := TRUE);

opResp   := fb.Ack(eRequester := TcForge.E_Requester.OPERATOR);
progResp := fb.Ack(eRequester := TcForge.E_Requester.PROG);

AssertEquals_DINT(
    Expected := TcForge.E_RpcMethodResponse.REJECTED_SOURCE_NOT_ALLOWED,
    Actual   := opResp,
    Message  := 'Source-locked alarm must reject OPERATOR Ack()');
AssertEquals_DINT(
    Expected := TcForge.E_RpcMethodResponse.ACCEPTED,
    Actual   := progResp,
    Message  := 'Source-locked alarm must still accept PROG Ack()');

TEST_FINISHED();
END_METHOD

METHOD AckWithNoLatchIsNoOp
VAR
    fb       : TcForge.FB_AlarmSimple;
    response : TcForge.E_RpcMethodResponse;
END_VAR
TEST('AckWithNoLatchIsNoOp');

fb.cfg.common.bEnable     := TRUE;
fb.cfg.common.bRequireAck := TRUE;

// Ack() before any latch exists is accepted (the requester validation
// passes) but must leave acked FALSE — there is nothing to mark acked.
fb(inpActive := FALSE);
response := fb.Ack(eRequester := TcForge.E_Requester.OPERATOR);
fb(inpActive := FALSE);

AssertEquals_DINT(
    Expected := TcForge.E_RpcMethodResponse.ACCEPTED,
    Actual   := response,
    Message  := 'Ack() with no latch returns ACCEPTED (validation passes)');
AssertFalse(
    Condition := fb.sts.acked,
    Message   := 'Ack() with no latch must NOT flip acked — there is no latch to ack');

TEST_FINISHED();
END_METHOD

END_FUNCTION_BLOCK

// ---- Tests/FB_AlarmLimit_Test.TcPOU
// Tests for FB_AlarmLimit — four-level (HiHi/Hi/Lo/LoLo) ladder built by
// composing FB_AlarmThreshold. FB_AlarmSimple_Test already covers the
// shared FB_AlarmBase contract, so this suite focuses on the composite
// behaviour that lives only here:
//   - per-direction threshold evaluation via bFailHigh / bFailLow
//   - flood suppression (HiHi hides Hi, LoLo hides Lo) on the rollup flags
//     while keeping the raw sub-statuses available
//   - severity aggregation (highest-active wins)
//   - anyActive is the OR of all four rollup flags
//   - Ack() cascades to every level
FUNCTION_BLOCK FB_AlarmLimit_Test EXTENDS TcUnit.FB_TestSuite

AllDisabledStaysSilent();
HiTripsAboveThreshold();
HiHiSuppressesHiOnRollup();
LoTripsBelowThreshold();
LoLoSuppressesLoOnRollup();
SeverityIsHighestActiveLevel();
AnyActiveReflectsRollup();
AckCascadesToEveryLevel();

// Helper: configure HiHi and Hi as a typical upper ladder. Keeps each
// test method short and consistent with the example PRG_Alarms wiring.
METHOD PRIVATE _ConfigureHiHi
VAR_IN_OUT
    fb : TcForge.FB_AlarmLimit;
END_VAR
fb.cfg.HiHi.common.bEnable     := TRUE;
fb.cfg.HiHi.common.bRequireAck := FALSE;
fb.cfg.HiHi.common.eSeverity   := TcForge.E_AlarmSeverity.CRITICAL;
fb.cfg.HiHi.fThreshold         := 110.0;
fb.cfg.HiHi.bFailHigh          := TRUE;

fb.cfg.Hi.common.bEnable     := TRUE;
fb.cfg.Hi.common.bRequireAck := FALSE;
fb.cfg.Hi.common.eSeverity   := TcForge.E_AlarmSeverity.WARNING;
fb.cfg.Hi.fThreshold         := 100.0;
fb.cfg.Hi.bFailHigh          := TRUE;
END_METHOD

// Helper: configure Lo and LoLo as a typical lower ladder.
METHOD PRIVATE _ConfigureLoLo
VAR_IN_OUT
    fb : TcForge.FB_AlarmLimit;
END_VAR
fb.cfg.Lo.common.bEnable     := TRUE;
fb.cfg.Lo.common.bRequireAck := FALSE;
fb.cfg.Lo.common.eSeverity   := TcForge.E_AlarmSeverity.WARNING;
fb.cfg.Lo.fThreshold         := 20.0;
fb.cfg.Lo.bFailLow           := TRUE;

fb.cfg.LoLo.common.bEnable     := TRUE;
fb.cfg.LoLo.common.bRequireAck := FALSE;
fb.cfg.LoLo.common.eSeverity   := TcForge.E_AlarmSeverity.CRITICAL;
fb.cfg.LoLo.fThreshold         := 10.0;
fb.cfg.LoLo.bFailLow           := TRUE;
END_METHOD

METHOD AllDisabledStaysSilent
VAR
    fb : TcForge.FB_AlarmLimit;
END_VAR
TEST('AllDisabledStaysSilent');

// Every level disabled; rollup flags and severity must stay quiet even
// when the process value is far outside every sensible band.
fb(inpPv := 500.0);

AssertFalse(
    Condition := fb.sts.anyActive,
    Message   := 'anyActive must be FALSE when every level is disabled');
AssertEquals_USINT(
    Expected := TcForge.E_AlarmSeverity.NONE,
    Actual   := fb.sts.eSeverity,
    Message  := 'eSeverity must be NONE when every level is disabled');

TEST_FINISHED();
END_METHOD

METHOD HiTripsAboveThreshold
VAR
    fb : TcForge.FB_AlarmLimit;
END_VAR
TEST('HiTripsAboveThreshold');

_ConfigureHiHi(fb := fb);

fb(inpPv := 105.0);  // above Hi (100), below HiHi (110)

AssertTrue(
    Condition := fb.sts.hiActive,
    Message   := 'Hi should trip when PV crosses its threshold');
AssertFalse(
    Condition := fb.sts.hiHiActive,
    Message   := 'HiHi should stay inactive while PV is below the HiHi threshold');

TEST_FINISHED();
END_METHOD

METHOD HiHiSuppressesHiOnRollup
VAR
    fb : TcForge.FB_AlarmLimit;
END_VAR
TEST('HiHiSuppressesHiOnRollup');

_ConfigureHiHi(fb := fb);

fb(inpPv := 115.0);  // above both Hi and HiHi

AssertTrue(
    Condition := fb.sts.hiHiActive,
    Message   := 'HiHi should trip when PV crosses its threshold');
AssertFalse(
    Condition := fb.sts.hiActive,
    Message   := 'Hi must be suppressed on the rollup while HiHi is active');
AssertTrue(
    Condition := fb.sts.Hi.active,
    Message   := 'Raw Hi sub-status must still expose the trip (forensics channel)');

TEST_FINISHED();
END_METHOD

METHOD LoTripsBelowThreshold
VAR
    fb : TcForge.FB_AlarmLimit;
END_VAR
TEST('LoTripsBelowThreshold');

_ConfigureLoLo(fb := fb);

fb(inpPv := 15.0);  // below Lo (20), above LoLo (10)

AssertTrue(
    Condition := fb.sts.loActive,
    Message   := 'Lo should trip when PV drops below its threshold');
AssertFalse(
    Condition := fb.sts.loLoActive,
    Message   := 'LoLo should stay inactive while PV is above the LoLo threshold');

TEST_FINISHED();
END_METHOD

METHOD LoLoSuppressesLoOnRollup
VAR
    fb : TcForge.FB_AlarmLimit;
END_VAR
TEST('LoLoSuppressesLoOnRollup');

_ConfigureLoLo(fb := fb);

fb(inpPv := 5.0);  // below both Lo and LoLo

AssertTrue(
    Condition := fb.sts.loLoActive,
    Message   := 'LoLo should trip when PV drops below its threshold');
AssertFalse(
    Condition := fb.sts.loActive,
    Message   := 'Lo must be suppressed on the rollup while LoLo is active');
AssertTrue(
    Condition := fb.sts.Lo.active,
    Message   := 'Raw Lo sub-status must still expose the trip (forensics channel)');

TEST_FINISHED();
END_METHOD

METHOD SeverityIsHighestActiveLevel
VAR
    fb : TcForge.FB_AlarmLimit;
END_VAR
TEST('SeverityIsHighestActiveLevel');

_ConfigureHiHi(fb := fb);

// PV between Hi and HiHi → only Hi active → severity = WARNING.
fb(inpPv := 105.0);
AssertEquals_USINT(
    Expected := TcForge.E_AlarmSeverity.WARNING,
    Actual   := fb.sts.eSeverity,
    Message  := 'Severity should be WARNING when only Hi is active');

// PV above HiHi → HiHi (CRITICAL) wins even though raw Hi still fires.
fb(inpPv := 115.0);
AssertEquals_USINT(
    Expected := TcForge.E_AlarmSeverity.CRITICAL,
    Actual   := fb.sts.eSeverity,
    Message  := 'Severity should be CRITICAL once HiHi engages');

TEST_FINISHED();
END_METHOD

METHOD AnyActiveReflectsRollup
VAR
    fb : TcForge.FB_AlarmLimit;
END_VAR
TEST('AnyActiveReflectsRollup');

_ConfigureHiHi(fb := fb);
_ConfigureLoLo(fb := fb);

fb(inpPv := 50.0);  // in the good band
AssertFalse(
    Condition := fb.sts.anyActive,
    Message   := 'anyActive should be FALSE while PV sits in the good band');

fb(inpPv := 115.0);
AssertTrue(
    Condition := fb.sts.anyActive,
    Message   := 'anyActive should be TRUE once any level trips');

fb(inpPv := 50.0);
AssertFalse(
    Condition := fb.sts.anyActive,
    Message   := 'anyActive should go back FALSE when PV returns to the good band (non-latching cfg)');

TEST_FINISHED();
END_METHOD

METHOD AckCascadesToEveryLevel
VAR
    fb       : TcForge.FB_AlarmLimit;
    response : TcForge.E_RpcMethodResponse;
END_VAR
TEST('AckCascadesToEveryLevel');

// Both Hi and HiHi latching — a PV spike into HiHi latches both raw
// sub-alarms. Ack() must cascade so every level releases on the next
// post-clear cycle.
fb.cfg.HiHi.common.bEnable     := TRUE;
fb.cfg.HiHi.common.bRequireAck := TRUE;
fb.cfg.HiHi.common.eSeverity   := TcForge.E_AlarmSeverity.CRITICAL;
fb.cfg.HiHi.fThreshold         := 110.0;
fb.cfg.HiHi.bFailHigh          := TRUE;

fb.cfg.Hi.common.bEnable     := TRUE;
fb.cfg.Hi.common.bRequireAck := TRUE;
fb.cfg.Hi.common.eSeverity   := TcForge.E_AlarmSeverity.WARNING;
fb.cfg.Hi.fThreshold         := 100.0;
fb.cfg.Hi.bFailHigh          := TRUE;

// Spike then recover.
fb(inpPv := 115.0);
fb(inpPv := 50.0);

AssertTrue(
    Condition := fb.sts.HiHi.active AND fb.sts.Hi.active,
    Message   := 'Precondition: both raw sub-alarms should be latched after the spike');

response := fb.Ack(eRequester := TcForge.E_Requester.OPERATOR);
fb(inpPv := 50.0);

AssertEquals_DINT(
    Expected := TcForge.E_RpcMethodResponse.ACCEPTED,
    Actual   := response,
    Message  := 'Composite Ack() should be accepted when at least one level accepts');
AssertFalse(
    Condition := fb.sts.HiHi.active,
    Message   := 'HiHi latch must release after cascaded Ack() + clear');
AssertFalse(
    Condition := fb.sts.Hi.active,
    Message   := 'Hi latch must release after cascaded Ack() + clear');
AssertFalse(
    Condition := fb.sts.anyActive,
    Message   := 'anyActive should return FALSE once every level releases');

TEST_FINISHED();
END_METHOD

END_FUNCTION_BLOCK

// ---- Tests/FB_DeviceBase_Test.TcPOU
// Tests for FB_DeviceBase — the shared base for every TcForge device FB.
// Driven through FB_DeviceBase_Probe (a test-only concrete child) because
// the base is ABSTRACT and the fault book-keeping API is PROTECTED.
//
// Coverage focuses on the contract every device inherits:
//   - diagnostics (IsFaulted / GetFaultCode / GetFaultString with virtual
//     dispatch through the child's ResolveFaultString)
//   - _Raise semantics: zero-code no-op, idempotent on code within an
//     episode, different code replaces the active fault
//   - _ClearFault wipes the active fault but preserves lastFault* for
//     the header so HMIs can still render what happened
//   - Reset() is always accepted from any requester — safety invariant
//   - _UpdateHeader() mirrors the active/last fault, source-lock, busy,
//     and ready state into ST_DeviceHeader_Sts
//   - LockSource() makes sourceLocked and forces ready FALSE
FUNCTION_BLOCK FB_DeviceBase_Test EXTENDS TcUnit.FB_TestSuite

FreshInstanceNotFaulted();
RaiseZeroCodeIsNoOp();
RaiseSetsActiveFaultAndResolvesString();
RaiseSameCodeIsIdempotent();
DifferentCodeReplacesActiveFault();
ClearFaultWipesActiveButKeepsLastFault();
ResetAlwaysAcceptedEvenFromOperatorWhileLocked();
HeaderMirrorsActiveFault();
HeaderReadyGoesFalseOnSourceLock();
HeaderReadyGoesFalseOnBusy();

METHOD FreshInstanceNotFaulted
VAR
    fb : FB_DeviceBase_Probe;
END_VAR
TEST('FreshInstanceNotFaulted');

AssertFalse(
    Condition := fb.IsFaulted(),
    Message   := 'Fresh device must not be faulted');
AssertEquals_DINT(
    Expected := 0,
    Actual   := fb.GetFaultCode(),
    Message  := 'Fresh device fault code should be 0');
AssertEquals_STRING(
    Expected := '',
    Actual   := fb.GetFaultString(),
    Message  := 'Fresh device fault string should be empty');

TEST_FINISHED();
END_METHOD

METHOD RaiseZeroCodeIsNoOp
VAR
    fb     : FB_DeviceBase_Probe;
    result : BOOL;
END_VAR
TEST('RaiseZeroCodeIsNoOp');

// code = 0 is the "no fault" sentinel; calling _Raise(0, ...) must never
// register a fault nor push a ring entry.
result := fb.ProbeRaise(code := 0, source := 'test', reason := 'should not register');

AssertFalse(
    Condition := result,
    Message   := '_Raise(0) must return FALSE (nothing was pushed)');
AssertFalse(
    Condition := fb.IsFaulted(),
    Message   := '_Raise(0) must not put the device into a faulted state');

TEST_FINISHED();
END_METHOD

METHOD RaiseSetsActiveFaultAndResolvesString
VAR
    fb     : FB_DeviceBase_Probe;
    result : BOOL;
END_VAR
TEST('RaiseSetsActiveFaultAndResolvesString');

result := fb.ProbeRaise(code := 42, source := 'step5', reason := 'motion timeout');

AssertTrue(
    Condition := result,
    Message   := '_Raise of a new non-zero code must return TRUE (ring entry pushed)');
AssertTrue(
    Condition := fb.IsFaulted(),
    Message   := 'IsFaulted should be TRUE after a raise');
AssertEquals_DINT(
    Expected := 42,
    Actual   := fb.GetFaultCode(),
    Message  := 'GetFaultCode should report the raised code');
AssertEquals_STRING(
    Expected := 'Motion timeout',
    Actual   := fb.GetFaultString(),
    Message  := 'GetFaultString should resolve via the child ResolveFaultString override');

TEST_FINISHED();
END_METHOD

METHOD RaiseSameCodeIsIdempotent
VAR
    fb         : FB_DeviceBase_Probe;
    firstCall  : BOOL;
    secondCall : BOOL;
END_VAR
TEST('RaiseSameCodeIsIdempotent');

// Cyclic callers often raise the same fault every scan until cleared.
// A second raise of the same non-zero code within one episode must be a
// no-op so the ring buffer doesn't flood.
firstCall  := fb.ProbeRaise(code := 42, source := 'step5', reason := 'first call');
secondCall := fb.ProbeRaise(code := 42, source := 'step5', reason := 'second call — ignored');

AssertTrue(
    Condition := firstCall,
    Message   := 'First _Raise of a code must return TRUE');
AssertFalse(
    Condition := secondCall,
    Message   := 'Repeat _Raise of the same code within an episode must return FALSE (no new ring entry)');
AssertEquals_DINT(
    Expected := 42,
    Actual   := fb.GetFaultCode(),
    Message  := 'Active fault must still be the first code after a repeated raise');

TEST_FINISHED();
END_METHOD

METHOD DifferentCodeReplacesActiveFault
VAR
    fb      : FB_DeviceBase_Probe;
    first   : BOOL;
    second  : BOOL;
END_VAR
TEST('DifferentCodeReplacesActiveFault');

// A progression like 'Timeout' -> 'LimitTripped' should preserve both in
// the ring; the second raise returns TRUE and becomes the active fault.
first  := fb.ProbeRaise(code := 42, source := 'step5', reason := 'motion timeout');
second := fb.ProbeRaise(code := 99, source := 'step5', reason := 'limit tripped');

AssertTrue(
    Condition := first AND second,
    Message   := 'Both raises of different codes must return TRUE');
AssertEquals_DINT(
    Expected := 99,
    Actual   := fb.GetFaultCode(),
    Message  := 'Active fault must be the most recent code');
AssertEquals_STRING(
    Expected := 'Limit tripped',
    Actual   := fb.GetFaultString(),
    Message  := 'GetFaultString must reflect the new active code');

TEST_FINISHED();
END_METHOD

METHOD ClearFaultWipesActiveButKeepsLastFault
VAR
    fb : FB_DeviceBase_Probe;
END_VAR
TEST('ClearFaultWipesActiveButKeepsLastFault');

fb.ProbeRaise(code := 42, source := 'step5', reason := 'motion timeout');
fb.ProbeClearFault();

AssertFalse(
    Condition := fb.IsFaulted(),
    Message   := '_ClearFault must drop IsFaulted to FALSE');
AssertEquals_DINT(
    Expected := 0,
    Actual   := fb.GetFaultCode(),
    Message  := 'Active fault code must be 0 after _ClearFault');

// Header must still preserve last-fault fields so the HMI can render
// "last fault: motion timeout".
fb.Refresh(stateString := 'IDLE', busy := FALSE);

AssertEquals_DINT(
    Expected := 42,
    Actual   := fb.header.lastFaultCode,
    Message  := 'header.lastFaultCode must preserve history after _ClearFault');
AssertEquals_STRING(
    Expected := 'Motion timeout',
    Actual   := fb.header.lastFaultString,
    Message  := 'header.lastFaultString must preserve the resolved text after _ClearFault');

TEST_FINISHED();
END_METHOD

METHOD ResetAlwaysAcceptedEvenFromOperatorWhileLocked
VAR
    fb       : FB_DeviceBase_Probe;
    response : TcForge.E_RpcMethodResponse;
END_VAR
TEST('ResetAlwaysAcceptedEvenFromOperatorWhileLocked');

// Safety invariant: Reset() is always accepted, regardless of source lock
// or active fault. No one should be locked out of clearing a fault.
fb.LockSource(bLock := TRUE);
fb.ProbeRaise(code := 42, source := 'step5', reason := 'motion timeout');

response := fb.Reset(eRequester := TcForge.E_Requester.OPERATOR);

AssertEquals_DINT(
    Expected := TcForge.E_RpcMethodResponse.ACCEPTED,
    Actual   := response,
    Message  := 'Reset() must be accepted from OPERATOR even while source-locked');
AssertFalse(
    Condition := fb.IsFaulted(),
    Message   := 'Reset() must clear the active fault');

TEST_FINISHED();
END_METHOD

METHOD HeaderMirrorsActiveFault
VAR
    fb : FB_DeviceBase_Probe;
END_VAR
TEST('HeaderMirrorsActiveFault');

fb.ProbeRaise(code := 99, source := 'limit_sw', reason := 'upper limit hit');
fb.Refresh(stateString := 'FAULTED', busy := FALSE);

AssertTrue(
    Condition := fb.header.faulted,
    Message   := 'header.faulted must be TRUE while a fault is active');
AssertFalse(
    Condition := fb.header.ready,
    Message   := 'header.ready must be FALSE while faulted');
AssertEquals_DINT(
    Expected := 99,
    Actual   := fb.header.faultCode,
    Message  := 'header.faultCode must mirror the active fault');
AssertEquals_STRING(
    Expected := 'Limit tripped',
    Actual   := fb.header.faultString,
    Message  := 'header.faultString must resolve via the child override');
AssertEquals_STRING(
    Expected := 'limit_sw',
    Actual   := fb.header.faultSource,
    Message  := 'header.faultSource must carry the raise() source');
AssertEquals_STRING(
    Expected := 'upper limit hit',
    Actual   := fb.header.faultReason,
    Message  := 'header.faultReason must carry the raise() reason');
AssertEquals_STRING(
    Expected := 'FAULTED',
    Actual   := fb.header.stateString,
    Message  := 'header.stateString must mirror the state string passed to _UpdateHeader');

TEST_FINISHED();
END_METHOD

METHOD HeaderReadyGoesFalseOnSourceLock
VAR
    fb : FB_DeviceBase_Probe;
END_VAR
TEST('HeaderReadyGoesFalseOnSourceLock');

fb.Refresh(stateString := 'IDLE', busy := FALSE);
AssertTrue(
    Condition := fb.header.ready,
    Message   := 'Precondition: an idle / unlocked / unfaulted device must be ready');

fb.LockSource(bLock := TRUE);
fb.Refresh(stateString := 'IDLE', busy := FALSE);

AssertTrue(
    Condition := fb.header.sourceLocked,
    Message   := 'header.sourceLocked must mirror LockSource(TRUE)');
AssertFalse(
    Condition := fb.header.ready,
    Message   := 'header.ready must be FALSE while source is locked');

TEST_FINISHED();
END_METHOD

METHOD HeaderReadyGoesFalseOnBusy
VAR
    fb : FB_DeviceBase_Probe;
END_VAR
TEST('HeaderReadyGoesFalseOnBusy');

fb.Refresh(stateString := 'MOVING', busy := TRUE);

AssertTrue(
    Condition := fb.header.busy,
    Message   := 'header.busy must mirror the busy flag passed to _UpdateHeader');
AssertFalse(
    Condition := fb.header.ready,
    Message   := 'header.ready must be FALSE while busy');

TEST_FINISHED();
END_METHOD

END_FUNCTION_BLOCK

// ---- POUs/FB_DeviceBase_Probe.TcPOU
// Test-only concrete child of FB_DeviceBase. Exposes the protected API
// (_Raise / _ClearFault / _AcceptCommand / _UpdateHeader) through public
// "Probe*" wrappers so FB_DeviceBase_Test can drive the base contract
// without a full device FB in the way. Also overrides ResolveFaultString
// so the tests can verify virtual dispatch.
//
// This FB lives in the Testing project on purpose — it is not part of the
// TcForge public surface.
FUNCTION_BLOCK FB_DeviceBase_Probe EXTENDS TcForge.FB_DeviceBase
VAR_OUTPUT
    header : TcForge.ST_DeviceHeader_Sts;
END_VAR

// Nothing cyclic — tests call the probe methods directly.

METHOD PUBLIC ProbeRaise : BOOL
VAR_INPUT
    code   : DINT;
    source : STRING(31);
    reason : STRING(79);
END_VAR
ProbeRaise := _Raise(code := code, source := source, reason := reason);
END_METHOD

METHOD PUBLIC ProbeClearFault
_ClearFault();
END_METHOD

METHOD PUBLIC ProbeAcceptCommand
VAR_INPUT
    eRequester : TcForge.E_Requester;
END_VAR
_AcceptCommand(eRequester := eRequester);
END_METHOD

// Populate the probe's own header struct via the protected _UpdateHeader.
METHOD PUBLIC Refresh
VAR_INPUT
    stateString : STRING(31);
    busy     : BOOL;
END_VAR
_UpdateHeader(
    header      := header,
    stateString := stateString,
    busy     := busy);
END_METHOD

// Minimal resolver so the tests can verify virtual dispatch through the
// base's GetFaultString() / _UpdateHeader() calls. Maps a few well-known
// codes; everything else returns empty (inherited default behaviour).
METHOD PROTECTED ResolveFaultString : STRING(79)
VAR_INPUT
    code : DINT;
END_VAR
CASE code OF
    42: ResolveFaultString := 'Motion timeout';
    99: ResolveFaultString := 'Limit tripped';
ELSE
    ResolveFaultString := '';
END_CASE;
END_METHOD

END_FUNCTION_BLOCK

// ---- Tests/FB_LPF_FirstOrder_IIR_Test.TcPOU
// Tests for FB_LPF_FirstOrder_IIR — exponential-smoothing low-pass filter.
// Pure math, no external coupling, so each test drives a fresh instance
// with deterministic samples and checks the output against the closed-
// form IIR recurrence:
//     alpha = dt / (tau + dt)
//     y[n]  = y[n-1] + alpha * (x[n] - y[n-1])
//
// Floating-point results are compared with a tolerance via AssertTrue on
// ABS(actual - expected); TcUnit's primitive AssertEquals_LREAL does not
// accept a delta.
FUNCTION_BLOCK FB_LPF_FirstOrder_IIR_Test EXTENDS TcUnit.FB_TestSuite
VAR CONSTANT
    TOL : LREAL := 1E-9;  // generous floating-point tolerance for LREAL math
END_VAR

ZeroDtBypassesFilterAndRaisesError();
ZeroTauBypassesFilterAndRaisesError();
FirstSampleMatchesIirRecurrence();
StateCarriesBetweenCalls();
ConvergesTowardInputOverManySamples();
ErrorClearsOnValidInputAfterBadInput();

METHOD ZeroDtBypassesFilterAndRaisesError
VAR
    fb : TcForge.FB_LPF_FirstOrder_IIR;
END_VAR
TEST('ZeroDtBypassesFilterAndRaisesError');

// dt <= 0 cannot drive the recurrence, so the filter must fall back to
// passthrough and surface bError so the caller can notice.
fb(fInput := 42.0, fDt := 0.0, fTau := 1.0);

AssertTrue(
    Condition := ABS(fb.fOutput - 42.0) < TOL,
    Message   := 'With fDt = 0 the filter must pass the input through unchanged');
AssertTrue(
    Condition := fb.bError,
    Message   := 'With fDt = 0 the filter must raise bError');

TEST_FINISHED();
END_METHOD

METHOD ZeroTauBypassesFilterAndRaisesError
VAR
    fb : TcForge.FB_LPF_FirstOrder_IIR;
END_VAR
TEST('ZeroTauBypassesFilterAndRaisesError');

fb(fInput := 7.5, fDt := 0.1, fTau := 0.0);

AssertTrue(
    Condition := ABS(fb.fOutput - 7.5) < TOL,
    Message   := 'With fTau = 0 the filter must pass the input through unchanged');
AssertTrue(
    Condition := fb.bError,
    Message   := 'With fTau = 0 the filter must raise bError');

TEST_FINISHED();
END_METHOD

METHOD FirstSampleMatchesIirRecurrence
VAR
    fb       : TcForge.FB_LPF_FirstOrder_IIR;
    expected : LREAL;
    alpha    : LREAL;
END_VAR
TEST('FirstSampleMatchesIirRecurrence');

// Fresh instance: _prevOutput_sync = 0. With input 10, dt 0.1, tau 1.0:
//   alpha = 0.1 / 1.1
//   y[0]  = 0 + alpha * (10 - 0) = alpha * 10
alpha    := 0.1 / 1.1;
expected := alpha * 10.0;

fb(fInput := 10.0, fDt := 0.1, fTau := 1.0);

AssertFalse(
    Condition := fb.bError,
    Message   := 'Valid dt / tau must clear bError');
AssertTrue(
    Condition := ABS(fb.fOutput - expected) < TOL,
    Message   := 'First sample must match the IIR recurrence against zero state');

TEST_FINISHED();
END_METHOD

METHOD StateCarriesBetweenCalls
VAR
    fb        : TcForge.FB_LPF_FirstOrder_IIR;
    alpha     : LREAL;
    y1        : LREAL;
    yExpected : LREAL;
END_VAR
TEST('StateCarriesBetweenCalls');

alpha := 0.1 / 1.1;

fb(fInput := 10.0, fDt := 0.1, fTau := 1.0);
y1 := fb.fOutput;

// Second sample: y[1] = y[0] + alpha * (10 - y[0])
yExpected := y1 + alpha * (10.0 - y1);

fb(fInput := 10.0, fDt := 0.1, fTau := 1.0);

AssertTrue(
    Condition := ABS(fb.fOutput - yExpected) < TOL,
    Message   := 'Second sample must fold the previous output through the IIR recurrence (state is preserved across calls)');

TEST_FINISHED();
END_METHOD

METHOD ConvergesTowardInputOverManySamples
VAR
    fb     : TcForge.FB_LPF_FirstOrder_IIR;
    target : LREAL := 10.0;
    i      : UDINT;
END_VAR
TEST('ConvergesTowardInputOverManySamples');

// 200 samples at dt = tau/20 is well past steady-state — the output must
// be within ~1e-3 of the input regardless of the exact alpha value.
FOR i := 1 TO 200 DO
    fb(fInput := target, fDt := 0.05, fTau := 1.0);
END_FOR;

AssertTrue(
    Condition := ABS(fb.fOutput - target) < 1E-3,
    Message   := 'After many samples the filter output must converge toward the input');

TEST_FINISHED();
END_METHOD

METHOD ErrorClearsOnValidInputAfterBadInput
VAR
    fb : TcForge.FB_LPF_FirstOrder_IIR;
END_VAR
TEST('ErrorClearsOnValidInputAfterBadInput');

// A bad sample raises the flag; the very next valid sample must clear it.
fb(fInput := 5.0, fDt := 0.0, fTau := 1.0);
AssertTrue(
    Condition := fb.bError,
    Message   := 'Precondition: bError should be TRUE after a bad sample');

fb(fInput := 5.0, fDt := 0.1, fTau := 1.0);
AssertFalse(
    Condition := fb.bError,
    Message   := 'bError must clear the cycle a valid sample lands');

TEST_FINISHED();
END_METHOD

END_FUNCTION_BLOCK

// ---- Tests/FB_DigitalOutput_Test.TcPOU
// Tests for FB_DigitalOutput. Focus is on the behavior the device exposes
// to callers and HMIs:
//
//   * command routing through F_ValidateRequester (source lock)
//   * request-vs-output bookkeeping (commanded always reflects the
//     latest intent, value always reflects the physical bit)
//   * debounce timers actually gating the output
//   * invert in Regular mode
//   * BAD quality holding the last-known-good output
//   * edge pulses being exactly one scan wide
//   * SinglePulse arming on rising edge and cancelling on commanded LOW
//
// Time-dependent behavior is covered by choosing timer values that either
// clamp to zero (instant fire) or stay effectively infinite for the test
// (T#1S), so a single cyclic call lands in the branch under test without
// waiting real time.
FUNCTION_BLOCK FB_DigitalOutput_Test EXTENDS TcUnit.FB_TestSuite

InitialStateReady();
SetOnFromProgDrivesOutputHigh();
SetOffAfterSetOnDrivesOutputLow();
SetOnAcceptedFromProgEvenWhenLocked();
SetOnRejectedFromOperatorWhenLocked();
DebounceOnBlocksOutputUntilElapsed();
DebounceOffHoldsOutputHighUntilElapsed();
InvertFlipsOutputInRegularMode();
BadQualityHoldsLastKnownGoodOutput();
StsCommandedMirrorsRequestEvenUnderBadQuality();
EdgePulsesAreOneScanWide();
SinglePulseFiresOnCommandAndCanBeCanceled();

METHOD InitialStateReady
VAR
    fb : TcForge.FB_DigitalOutput;
END_VAR
TEST('InitialStateReady');

// Fresh instance + one good-quality cycle: no commands issued, no faults
// raised, output dead.
fb(inpQuality := TcForge.E_IO_Quality.GOOD);

AssertFalse(
    Condition := fb.sts.value,
    Message   := 'Fresh instance must start with physical output LOW');
AssertFalse(
    Condition := fb.sts.commanded,
    Message   := 'Fresh instance must start with commanded request LOW');
AssertFalse(
    Condition := fb.sts.header.faulted,
    Message   := 'Fresh instance must not be faulted');
AssertTrue(
    Condition := fb.sts.header.ready,
    Message   := 'Fresh instance must report ready TRUE (no fault, not busy, not locked)');
AssertFalse(
    Condition := fb.sts.header.sourceLocked,
    Message   := 'Fresh instance must not be source-locked');

TEST_FINISHED();
END_METHOD

METHOD SetOnFromProgDrivesOutputHigh
VAR
    fb     : TcForge.FB_DigitalOutput;
    resp   : TcForge.E_RpcMethodResponse;
END_VAR
TEST('SetOnFromProgDrivesOutputHigh');

// Default cfg: no debounce (PT = T#0MS), Regular mode, no invert.
// A single SetOn + one cycle should flush straight through to the
// physical output.
resp := fb.SetOn(eRequester := TcForge.E_Requester.PROG);
fb(inpQuality := TcForge.E_IO_Quality.GOOD);

AssertEquals_DINT(
    Expected := TcForge.E_RpcMethodResponse.ACCEPTED,
    Actual   := resp,
    Message  := 'SetOn from PROG on a fresh instance must be ACCEPTED');
AssertTrue(
    Condition := fb.sts.value,
    Message   := 'Regular mode with no debounce must flush SetOn to the physical output in one cycle');
AssertTrue(
    Condition := fb.sts.commanded,
    Message   := 'commanded must reflect the accepted SetOn request');

TEST_FINISHED();
END_METHOD

METHOD SetOffAfterSetOnDrivesOutputLow
VAR
    fb   : TcForge.FB_DigitalOutput;
    resp : TcForge.E_RpcMethodResponse;
END_VAR
TEST('SetOffAfterSetOnDrivesOutputLow');

fb.SetOn(eRequester := TcForge.E_Requester.PROG);
fb(inpQuality := TcForge.E_IO_Quality.GOOD);

resp := fb.SetOff(eRequester := TcForge.E_Requester.PROG);
fb(inpQuality := TcForge.E_IO_Quality.GOOD);

AssertEquals_DINT(
    Expected := TcForge.E_RpcMethodResponse.ACCEPTED,
    Actual   := resp,
    Message  := 'SetOff from PROG must be ACCEPTED');
AssertFalse(
    Condition := fb.sts.value,
    Message   := 'SetOff must drop the physical output LOW in one cycle with no debounce');
AssertFalse(
    Condition := fb.sts.commanded,
    Message   := 'commanded must follow the latest SetOff request');

TEST_FINISHED();
END_METHOD

METHOD SetOnAcceptedFromProgEvenWhenLocked
VAR
    fb   : TcForge.FB_DigitalOutput;
    resp : TcForge.E_RpcMethodResponse;
END_VAR
TEST('SetOnAcceptedFromProgEvenWhenLocked');

// bSourceLockedToProg is meant to gate OPERATOR; PROG must always get
// through so the program can still drive the output after locking out the
// operator.
fb.LockSource(bLock := TRUE);
resp := fb.SetOn(eRequester := TcForge.E_Requester.PROG);
fb(inpQuality := TcForge.E_IO_Quality.GOOD);

AssertEquals_DINT(
    Expected := TcForge.E_RpcMethodResponse.ACCEPTED,
    Actual   := resp,
    Message  := 'PROG requester must be accepted even with source-lock active');
AssertTrue(
    Condition := fb.sts.value,
    Message   := 'Accepted SetOn from PROG must still drive the physical output');
AssertTrue(
    Condition := fb.sts.header.sourceLocked,
    Message   := 'header must reflect source-lock state');

TEST_FINISHED();
END_METHOD

METHOD SetOnRejectedFromOperatorWhenLocked
VAR
    fb   : TcForge.FB_DigitalOutput;
    resp : TcForge.E_RpcMethodResponse;
END_VAR
TEST('SetOnRejectedFromOperatorWhenLocked');

fb.LockSource(bLock := TRUE);
resp := fb.SetOn(eRequester := TcForge.E_Requester.OPERATOR);
fb(inpQuality := TcForge.E_IO_Quality.GOOD);

AssertEquals_DINT(
    Expected := TcForge.E_RpcMethodResponse.REJECTED_SOURCE_NOT_ALLOWED,
    Actual   := resp,
    Message  := 'OPERATOR requester must be rejected while source-locked');
AssertFalse(
    Condition := fb.sts.value,
    Message   := 'Rejected SetOn must not touch the physical output');
AssertFalse(
    Condition := fb.sts.commanded,
    Message   := 'Rejected SetOn must not update commanded');

TEST_FINISHED();
END_METHOD

METHOD DebounceOnBlocksOutputUntilElapsed
VAR
    fb : TcForge.FB_DigitalOutput;
END_VAR
TEST('DebounceOnBlocksOutputUntilElapsed');

// debounceOn = T#1S — far longer than this synchronous test will run,
// so _tonOn.Q must still be FALSE when we check: the output must be held
// LOW while the debounce hasn't elapsed.
fb.cfg.debounceOn := T#1S;
fb.SetOn(eRequester := TcForge.E_Requester.PROG);
fb(inpQuality := TcForge.E_IO_Quality.GOOD);

AssertTrue(
    Condition := fb.sts.commanded,
    Message   := 'commanded must reflect the request immediately (debounce gates the output, not the request)');
AssertFalse(
    Condition := fb.sts.value,
    Message   := 'debounceOn must hold the physical output LOW until the TON elapses');

TEST_FINISHED();
END_METHOD

METHOD DebounceOffHoldsOutputHighUntilElapsed
VAR
    fb : TcForge.FB_DigitalOutput;
END_VAR
TEST('DebounceOffHoldsOutputHighUntilElapsed');

// debounceOn stays at 0 so the output flushes HIGH immediately. The
// OFF-debounce (T#1S) then holds it HIGH even after SetOff, until TOF.Q
// falls — which it will not inside this synchronous test.
fb.cfg.debounceOff := T#1S;
fb.SetOn(eRequester := TcForge.E_Requester.PROG);
fb(inpQuality := TcForge.E_IO_Quality.GOOD);

AssertTrue(
    Condition := fb.sts.value,
    Message   := 'Precondition: SetOn with zero ON-debounce must flush HIGH');

fb.SetOff(eRequester := TcForge.E_Requester.PROG);
fb(inpQuality := TcForge.E_IO_Quality.GOOD);

AssertFalse(
    Condition := fb.sts.commanded,
    Message   := 'commanded must follow the SetOff request regardless of debounce');
AssertTrue(
    Condition := fb.sts.value,
    Message   := 'debounceOff must hold the physical output HIGH until the TOF expires');

TEST_FINISHED();
END_METHOD

METHOD InvertFlipsOutputInRegularMode
VAR
    fb : TcForge.FB_DigitalOutput;
END_VAR
TEST('InvertFlipsOutputInRegularMode');

// Active-low actuator: invert means "commanded ON -> physical LOW".
fb.cfg.invert := TRUE;
fb.SetOn(eRequester := TcForge.E_Requester.PROG);
fb(inpQuality := TcForge.E_IO_Quality.GOOD);

AssertTrue(
    Condition := fb.sts.commanded,
    Message   := 'commanded must reflect logical intent, not inverted physical output');
AssertFalse(
    Condition := fb.sts.value,
    Message   := 'invert must flip HIGH intent into a LOW physical output');

fb.SetOff(eRequester := TcForge.E_Requester.PROG);
fb(inpQuality := TcForge.E_IO_Quality.GOOD);

AssertFalse(
    Condition := fb.sts.commanded,
    Message   := 'commanded must follow SetOff regardless of invert');
AssertTrue(
    Condition := fb.sts.value,
    Message   := 'invert must flip LOW intent into a HIGH physical output');

TEST_FINISHED();
END_METHOD

METHOD BadQualityHoldsLastKnownGoodOutput
VAR
    fb : TcForge.FB_DigitalOutput;
END_VAR
TEST('BadQualityHoldsLastKnownGoodOutput');
fb.cfg.holdOnBadQuality := TRUE;

// Establish HIGH under GOOD quality.
fb.SetOn(eRequester := TcForge.E_Requester.PROG);
fb(inpQuality := TcForge.E_IO_Quality.GOOD);
AssertTrue(
    Condition := fb.sts.value,
    Message   := 'Precondition: SetOn under GOOD quality must drive HIGH');

// Now drop to BAD and try to SetOff. The hardware write must be skipped
// so the actuator stays in its last-known-good state.
fb.SetOff(eRequester := TcForge.E_Requester.PROG);
fb(inpQuality := TcForge.E_IO_Quality.BAD);

AssertTrue(
    Condition := fb.sts.value,
    Message   := 'BAD quality must hold the last-known-good physical output (no hardware write)');
AssertEquals_USINT(
    Expected := TcForge.E_IO_Quality.BAD,
    Actual   := fb.sts.quality,
    Message  := 'quality must surface the BAD tag to downstream consumers');

TEST_FINISHED();
END_METHOD

METHOD StsCommandedMirrorsRequestEvenUnderBadQuality
VAR
    fb : TcForge.FB_DigitalOutput;
END_VAR
TEST('StsCommandedMirrorsRequestEvenUnderBadQuality');
fb.cfg.holdOnBadQuality := TRUE;

// Even when the hardware write is vetoed by quality, commanded must
// still echo the live request so HMIs can show "operator asked for OFF
// but the output is held HIGH because quality is BAD".
fb.SetOn(eRequester := TcForge.E_Requester.PROG);
fb(inpQuality := TcForge.E_IO_Quality.GOOD);
fb.SetOff(eRequester := TcForge.E_Requester.PROG);
fb(inpQuality := TcForge.E_IO_Quality.BAD);

AssertFalse(
    Condition := fb.sts.commanded,
    Message   := 'commanded must reflect the current request even when BAD quality blocks the hardware write');
AssertTrue(
    Condition := fb.sts.value,
    Message   := 'value must still show the held physical output');

TEST_FINISHED();
END_METHOD

METHOD EdgePulsesAreOneScanWide
VAR
    fb : TcForge.FB_DigitalOutput;
END_VAR
TEST('EdgePulsesAreOneScanWide');

// Rising-edge pulse appears the cycle the physical output goes HIGH and
// is gone the next cycle.
fb.SetOn(eRequester := TcForge.E_Requester.PROG);
fb(inpQuality := TcForge.E_IO_Quality.GOOD);
AssertTrue(
    Condition := fb.sts.risingEdge,
    Message   := 'risingEdge must fire on the cycle the physical output goes HIGH');
AssertFalse(
    Condition := fb.sts.fallingEdge,
    Message   := 'fallingEdge must stay LOW on a rising edge cycle');

fb(inpQuality := TcForge.E_IO_Quality.GOOD);
AssertFalse(
    Condition := fb.sts.risingEdge,
    Message   := 'risingEdge must be exactly one scan wide');

// Falling edge on the way back down.
fb.SetOff(eRequester := TcForge.E_Requester.PROG);
fb(inpQuality := TcForge.E_IO_Quality.GOOD);
AssertTrue(
    Condition := fb.sts.fallingEdge,
    Message   := 'fallingEdge must fire on the cycle the physical output goes LOW');

fb(inpQuality := TcForge.E_IO_Quality.GOOD);
AssertFalse(
    Condition := fb.sts.fallingEdge,
    Message   := 'fallingEdge must be exactly one scan wide');

TEST_FINISHED();
END_METHOD

METHOD SinglePulseFiresOnCommandAndCanBeCanceled
VAR
    fb : TcForge.FB_DigitalOutput;
END_VAR
TEST('SinglePulseFiresOnCommandAndCanBeCanceled');

// SinglePulse with a long pulse width (T#10S) so the _tonPulseOn.Q
// stays FALSE inside this synchronous test and we observe the pulse
// while it is active.
fb.cfg.mode    := TcForge.E_DigitalOutput_Mode.SinglePulse;
fb.cfg.pulseOn := T#10S;

fb.SetOn(eRequester := TcForge.E_Requester.PROG);
fb(inpQuality := TcForge.E_IO_Quality.GOOD);

AssertTrue(
    Condition := fb.sts.value,
    Message   := 'SinglePulse must arm on the commanded rising edge and drive HIGH while active');

// Commanded LOW must cancel the pulse early — operator safety shortcut.
fb.SetOff(eRequester := TcForge.E_Requester.PROG);
fb(inpQuality := TcForge.E_IO_Quality.GOOD);

AssertFalse(
    Condition := fb.sts.value,
    Message   := 'SetOff must cancel an in-flight SinglePulse immediately');

TEST_FINISHED();
END_METHOD

END_FUNCTION_BLOCK

// ---- Tests/FB_DigitalInput_Test.TcPOU
// Tests exercise the public input/output and command contracts.
FUNCTION_BLOCK FB_DigitalInput_Test EXTENDS TcUnit.FB_TestSuite

InitialStateClean();
RawSignalPassthroughWithNoDebounce();
InvertFlipsDebouncedValueNotRaw();
RisingEdgePulseOneScan();
FallingEdgePulseOneScan();
DebounceOnBlocksRisingEdgeUntilElapsed();
DebounceOffHoldsSignalHighAfterRawGoesLow();
BadQualityHoldsLastRawValue();
QualityTagSurfacesInStatus();
ClampedQualityReadsAsGood();

METHOD InitialStateClean
VAR
    fb : TcForge.FB_DigitalInput;
END_VAR
TEST('InitialStateClean');

fb(inpQuality := TcForge.E_IO_Quality.GOOD);

AssertFalse(
    Condition := fb.sts.value,
    Message   := 'Fresh instance must read LOW when the physical input is LOW');
AssertFalse(
    Condition := fb.sts.rawValue,
    Message   := 'Fresh instance must report the raw input LOW');
AssertFalse(
    Condition := fb.sts.risingEdge,
    Message   := 'Fresh instance must not emit a spurious rising edge');
AssertFalse(
    Condition := fb.sts.fallingEdge,
    Message   := 'Fresh instance must not emit a spurious falling edge');
AssertFalse(
    Condition := fb.sts.header.faulted,
    Message   := 'Fresh instance must not be faulted');

TEST_FINISHED();
END_METHOD

METHOD RawSignalPassthroughWithNoDebounce
VAR
    fb : TcForge.FB_DigitalInput;
END_VAR
TEST('RawSignalPassthroughWithNoDebounce');

// Default cfg: no debounce, no invert. Raw hardware bit flushes through
// to value in one cycle.
fb.inSignal := TRUE;
fb(inpQuality := TcForge.E_IO_Quality.GOOD);

AssertTrue(
    Condition := fb.sts.rawValue,
    Message   := 'rawValue must echo the hardware bit under GOOD quality');
AssertTrue(
    Condition := fb.sts.value,
    Message   := 'With no debounce and no invert the conditioned value must match the raw bit');

TEST_FINISHED();
END_METHOD

METHOD InvertFlipsDebouncedValueNotRaw
VAR
    fb : TcForge.FB_DigitalInput;
END_VAR
TEST('InvertFlipsDebouncedValueNotRaw');

// Invert must apply to the debounced / published value but the raw
// reading should stay true-to-the-wire so troubleshooters can see what
// the hardware is actually doing.
fb.cfg.invert := TRUE;
fb.inSignal := TRUE;
fb(inpQuality := TcForge.E_IO_Quality.GOOD);

AssertTrue(
    Condition := fb.sts.rawValue,
    Message   := 'rawValue must echo the wire value independent of invert');
AssertFalse(
    Condition := fb.sts.value,
    Message   := 'invert must flip the conditioned value (active-low sensor semantics)');

TEST_FINISHED();
END_METHOD

METHOD RisingEdgePulseOneScan
VAR
    fb : TcForge.FB_DigitalInput;
END_VAR
TEST('RisingEdgePulseOneScan');

fb.inSignal := FALSE;
fb(inpQuality := TcForge.E_IO_Quality.GOOD);

fb.inSignal := TRUE;
fb(inpQuality := TcForge.E_IO_Quality.GOOD);
AssertTrue(
    Condition := fb.sts.risingEdge,
    Message   := 'risingEdge must fire on the cycle the debounced value goes HIGH');

fb(inpQuality := TcForge.E_IO_Quality.GOOD);
AssertFalse(
    Condition := fb.sts.risingEdge,
    Message   := 'risingEdge must clear the very next cycle — edges are one-scan pulses');

TEST_FINISHED();
END_METHOD

METHOD FallingEdgePulseOneScan
VAR
    fb : TcForge.FB_DigitalInput;
END_VAR
TEST('FallingEdgePulseOneScan');

fb.inSignal := TRUE;
fb(inpQuality := TcForge.E_IO_Quality.GOOD);

fb.inSignal := FALSE;
fb(inpQuality := TcForge.E_IO_Quality.GOOD);
AssertTrue(
    Condition := fb.sts.fallingEdge,
    Message   := 'fallingEdge must fire on the cycle the debounced value goes LOW');

fb(inpQuality := TcForge.E_IO_Quality.GOOD);
AssertFalse(
    Condition := fb.sts.fallingEdge,
    Message   := 'fallingEdge must clear the very next cycle');

TEST_FINISHED();
END_METHOD

METHOD DebounceOnBlocksRisingEdgeUntilElapsed
VAR
    fb : TcForge.FB_DigitalInput;
END_VAR
TEST('DebounceOnBlocksRisingEdgeUntilElapsed');

// debounceOn = T#1S — the _tonOn.Q won't fire inside this test frame.
fb.cfg.debounceOn := T#1S;
fb.inSignal := TRUE;
fb(inpQuality := TcForge.E_IO_Quality.GOOD);

AssertTrue(
    Condition := fb.sts.rawValue,
    Message   := 'rawValue must still show the raw bit — debounce gates the conditioned value, not the raw view');
AssertFalse(
    Condition := fb.sts.value,
    Message   := 'debounceOn must hold value LOW until the TON elapses');
AssertFalse(
    Condition := fb.sts.risingEdge,
    Message   := 'No rising edge must be emitted while debounce is pending');

TEST_FINISHED();
END_METHOD

METHOD DebounceOffHoldsSignalHighAfterRawGoesLow
VAR
    fb : TcForge.FB_DigitalInput;
END_VAR
TEST('DebounceOffHoldsSignalHighAfterRawGoesLow');

// debounceOff = T#1S. With debounceOn still 0 we latch the
// debounced signal HIGH immediately, then flip the raw bit LOW and
// expect the TOF to hold the debounced value HIGH.
fb.cfg.debounceOff := T#1S;
fb.inSignal := TRUE;
fb(inpQuality := TcForge.E_IO_Quality.GOOD);
AssertTrue(
    Condition := fb.sts.value,
    Message   := 'Precondition: raw HIGH with zero ON-debounce must latch the debounced value HIGH');

fb.inSignal := FALSE;
fb(inpQuality := TcForge.E_IO_Quality.GOOD);

AssertFalse(
    Condition := fb.sts.rawValue,
    Message   := 'rawValue must immediately mirror the wire going LOW');
AssertTrue(
    Condition := fb.sts.value,
    Message   := 'debounceOff must hold the debounced value HIGH until the TOF expires');
AssertFalse(
    Condition := fb.sts.fallingEdge,
    Message   := 'No falling edge must be emitted while the OFF-debounce is pending');

TEST_FINISHED();
END_METHOD

METHOD BadQualityHoldsLastRawValue
VAR
    fb : TcForge.FB_DigitalInput;
END_VAR
TEST('BadQualityHoldsLastRawValue');

// Latch a known-good HIGH reading.
fb.inSignal := TRUE;
fb(inpQuality := TcForge.E_IO_Quality.GOOD);
AssertTrue(
    Condition := fb.sts.rawValue,
    Message   := 'Precondition: under GOOD quality rawValue mirrors the wire');

// Simulate wire break: the underlying bit flips FALSE but quality is BAD.
// The FB must ignore the glitchy reading and hold the last-known-good raw.
fb.inSignal := FALSE;
fb(inpQuality := TcForge.E_IO_Quality.BAD);

AssertTrue(
    Condition := fb.sts.rawValue,
    Message   := 'BAD quality must freeze rawValue at the last known-good reading');
AssertEquals_USINT(
    Expected := TcForge.E_IO_Quality.BAD,
    Actual   := fb.sts.quality,
    Message  := 'quality must surface the BAD tag so downstream consumers can react');

TEST_FINISHED();
END_METHOD

METHOD QualityTagSurfacesInStatus
VAR
    fb : TcForge.FB_DigitalInput;
END_VAR
TEST('QualityTagSurfacesInStatus');

// UNKNOWN -> BAD -> GOOD must each land in sts.quality unchanged so
// the HMI can display the exact tag the caller supplied.
fb(inpQuality := TcForge.E_IO_Quality.UNKNOWN);
AssertEquals_USINT(
    Expected := TcForge.E_IO_Quality.UNKNOWN,
    Actual   := fb.sts.quality,
    Message  := 'quality must surface UNKNOWN unchanged');

fb(inpQuality := TcForge.E_IO_Quality.BAD);
AssertEquals_USINT(
    Expected := TcForge.E_IO_Quality.BAD,
    Actual   := fb.sts.quality,
    Message  := 'quality must surface BAD unchanged');

fb(inpQuality := TcForge.E_IO_Quality.GOOD);
AssertEquals_USINT(
    Expected := TcForge.E_IO_Quality.GOOD,
    Actual   := fb.sts.quality,
    Message  := 'quality must surface GOOD unchanged');

TEST_FINISHED();
END_METHOD

METHOD ClampedQualityReadsAsGood
VAR
    fb : TcForge.FB_DigitalInput;
END_VAR
TEST('ClampedQualityReadsAsGood');

// The quality gate treats GOOD and CLAMPED as "trust the raw reading".
// CLAMPED is meant for analog signals that hit a scaling limit — for a
// digital input it has to behave the same as GOOD so a wrapper that
// passes CLAMPED through doesn't accidentally freeze the reading.
fb.inSignal := TRUE;
fb(inpQuality := TcForge.E_IO_Quality.CLAMPED);

AssertTrue(
    Condition := fb.sts.rawValue,
    Message   := 'CLAMPED quality must be treated like GOOD for raw readings');
AssertTrue(
    Condition := fb.sts.value,
    Message   := 'CLAMPED quality must not freeze the conditioned value');
AssertEquals_USINT(
    Expected := TcForge.E_IO_Quality.CLAMPED,
    Actual   := fb.sts.quality,
    Message  := 'quality must still surface CLAMPED so consumers know the raw came from a clamped source');

TEST_FINISHED();
END_METHOD

END_FUNCTION_BLOCK

// ---- Tests/FB_TwoPosActuator_Test.TcPOU
// Tests exercise the public input/output and command contracts.
FUNCTION_BLOCK FB_TwoPosActuator_Test EXTENDS TcUnit.FB_TestSuite

InitialStateIsUndefined();
UndefinedBecomesAdvancedOnFeedback();
UndefinedBecomesRetractedOnFeedback();
UndefinedFaultsWhenBothFeedbacksAssertSimultaneously();
AdvanceCommandDrivesStateToAdvancing();
AdvanceAtPositionRearms();
AdvanceRejectedWhenPermissiveNotMet();
AdvanceRejectedFromOperatorWhileSourceLocked();
AdvancingCompletesOnAdvancedFeedback();
AdvancingFaultsOnBothFeedback();
AdvancedFaultsOnLostFeedback();
RetractFromAdvancedDrivesRetracting();
AbortAlwaysAcceptedAndReturnsToUndefined();
ResetClearsFaultAndReturnsToUndefined();
HeaderBusyMirrorsMovingState();

METHOD InitialStateIsUndefined
VAR
    fb : TcForge.FB_TwoPosActuator;
END_VAR
TEST('InitialStateIsUndefined');

// No feedbacks, one cycle. currentState init is Undefined and the body
// only transitions out when a single feedback asserts.
fb();

AssertEquals_DINT(
    Expected := TcForge.E_TwoPosActuator_State.Undefined,
    Actual   := fb.sts.state,
    Message  := 'Fresh instance with no feedbacks must stay in Undefined');
AssertFalse(
    Condition := fb.outAdvance,
    Message   := 'Undefined state must de-energize outValveAdvance');
AssertFalse(
    Condition := fb.outRetract,
    Message   := 'Undefined state must de-energize outValveRetract');
AssertFalse(
    Condition := fb.sts.header.faulted,
    Message   := 'Fresh instance must not be faulted');

TEST_FINISHED();
END_METHOD

METHOD UndefinedBecomesAdvancedOnFeedback
VAR
    fb : TcForge.FB_TwoPosActuator;
END_VAR
TEST('UndefinedBecomesAdvancedOnFeedback');

// Simulate a device that was already at the advanced end-stop on boot.
fb.inAdvanced := TRUE;
fb();

AssertEquals_DINT(
    Expected := TcForge.E_TwoPosActuator_State.Advanced,
    Actual   := fb.sts.state,
    Message  := 'Undefined must latch to Advanced when only inFbkAdvanced is TRUE');
AssertTrue(
    Condition := fb.sts.advanced,
    Message   := 'advanced must follow the resolved state');
AssertFalse(
    Condition := fb.sts.retracted,
    Message   := 'retracted must be FALSE when Advanced');

TEST_FINISHED();
END_METHOD

METHOD UndefinedBecomesRetractedOnFeedback
VAR
    fb : TcForge.FB_TwoPosActuator;
END_VAR
TEST('UndefinedBecomesRetractedOnFeedback');

fb.inRetracted := TRUE;
fb();

AssertEquals_DINT(
    Expected := TcForge.E_TwoPosActuator_State.Retracted,
    Actual   := fb.sts.state,
    Message  := 'Undefined must latch to Retracted when only inFbkRetracted is TRUE');
AssertTrue(
    Condition := fb.sts.retracted,
    Message   := 'retracted must follow the resolved state');
AssertFalse(
    Condition := fb.sts.advanced,
    Message   := 'advanced must be FALSE when Retracted');

TEST_FINISHED();
END_METHOD

METHOD UndefinedFaultsWhenBothFeedbacksAssertSimultaneously
VAR
    fb : TcForge.FB_TwoPosActuator;
END_VAR
TEST('UndefinedFaultsWhenBothFeedbacksAssertSimultaneously');

// A physically impossible sensor state — both end-stops asserted. The FB
// must trip to Fault with BothFeedbackOn instead of silently picking
// one branch.
fb.inAdvanced := TRUE;
fb.inRetracted := TRUE;
fb();

AssertEquals_DINT(
    Expected := TcForge.E_TwoPosActuator_State.Fault,
    Actual   := fb.sts.state,
    Message  := 'Both feedbacks simultaneously must drive state to Fault');
AssertTrue(
    Condition := fb.sts.header.faulted,
    Message   := 'header must report faulted when both feedbacks assert');
AssertEquals_DINT(
    Expected := TcForge.E_TwoPosActuator_Fault.BothFeedbackOn,
    Actual   := fb.sts.header.faultCode,
    Message  := 'Active fault code must be BothFeedbackOn');
AssertFalse(
    Condition := fb.outAdvance,
    Message   := 'Fault state must de-energize outValveAdvance');
AssertFalse(
    Condition := fb.outRetract,
    Message   := 'Fault state must de-energize outValveRetract');

TEST_FINISHED();
END_METHOD

METHOD AdvanceCommandDrivesStateToAdvancing
VAR
    fb   : TcForge.FB_TwoPosActuator;
    resp : TcForge.E_RpcMethodResponse;
END_VAR
TEST('AdvanceCommandDrivesStateToAdvancing');

// Start from Retracted (single known end-stop) — the canonical starting
// point before an Advance command.
fb.inRetracted := TRUE;
fb();
AssertEquals_DINT(
    Expected := TcForge.E_TwoPosActuator_State.Retracted,
    Actual   := fb.sts.state,
    Message  := 'Precondition: feedback-only start must settle to Retracted');

// Drop the retracted feedback first (simulates real physical travel) so
// the Advancing branch isn't racing against a lost-feedback trip.
fb.inRetracted := FALSE;

resp := fb.Advance(eRequester := TcForge.E_Requester.PROG);
fb();

AssertEquals_DINT(
    Expected := TcForge.E_RpcMethodResponse.ACCEPTED,
    Actual   := resp,
    Message  := 'Advance from PROG in Retracted must be ACCEPTED');
AssertEquals_DINT(
    Expected := TcForge.E_TwoPosActuator_State.Advancing,
    Actual   := fb.sts.state,
    Message  := 'Accepted Advance must transition state to Advancing');
AssertTrue(
    Condition := fb.outAdvance,
    Message   := 'Advancing state must energize outValveAdvance');
AssertFalse(
    Condition := fb.outRetract,
    Message   := 'Advancing state must NOT energize outValveRetract');
AssertTrue(
    Condition := fb.sts.moving,
    Message   := 'moving must flag the Advancing transit');

TEST_FINISHED();
END_METHOD

METHOD AdvanceAtPositionRearms
VAR
    fb   : TcForge.FB_TwoPosActuator;
    resp : TcForge.E_RpcMethodResponse;
END_VAR
TEST('AdvanceAtPositionRearms');

fb.inAdvanced := TRUE;
fb();
AssertEquals_DINT(
    Expected := TcForge.E_TwoPosActuator_State.Advanced,
    Actual   := fb.sts.state,
    Message  := 'Precondition: must be Advanced before rearming');

resp := fb.Advance(eRequester := TcForge.E_Requester.PROG);

AssertEquals_DINT(
    Expected := TcForge.E_RpcMethodResponse.ACCEPTED,
    Actual   := resp,
    Message  := 'Advance at known position explicitly rearms the device');

TEST_FINISHED();
END_METHOD

METHOD AdvanceRejectedWhenPermissiveNotMet
VAR
    fb   : TcForge.FB_TwoPosActuator;
    resp : TcForge.E_RpcMethodResponse;
END_VAR
TEST('AdvanceRejectedWhenPermissiveNotMet');

// Force the advance permissive to fail. One cycle is enough to let
// advancePermissives refresh sts.bOK to FALSE before we call Advance.
fb.MapAdvanceCondition(bitIndex := 0, bGood := FALSE);
fb();
fb.inRetracted := FALSE;

resp := fb.Advance(eRequester := TcForge.E_Requester.PROG);

AssertEquals_DINT(
    Expected := TcForge.E_RpcMethodResponse.REJECTED_PERMISSIVE_NOT_MET,
    Actual   := resp,
    Message  := 'Advance must be rejected when advancePermissives.sts.bOK is FALSE');

TEST_FINISHED();
END_METHOD

METHOD AdvanceRejectedFromOperatorWhileSourceLocked
VAR
    fb   : TcForge.FB_TwoPosActuator;
    resp : TcForge.E_RpcMethodResponse;
END_VAR
TEST('AdvanceRejectedFromOperatorWhileSourceLocked');

fb.LockSource(bLock := TRUE);
resp := fb.Advance(eRequester := TcForge.E_Requester.OPERATOR);

AssertEquals_DINT(
    Expected := TcForge.E_RpcMethodResponse.REJECTED_SOURCE_NOT_ALLOWED,
    Actual   := resp,
    Message  := 'OPERATOR must be rejected while source-locked');

TEST_FINISHED();
END_METHOD

METHOD AdvancingCompletesOnAdvancedFeedback
VAR
    fb : TcForge.FB_TwoPosActuator;
END_VAR
TEST('AdvancingCompletesOnAdvancedFeedback');

// One warmup cycle so advancePermissives refreshes sts.bOK to TRUE
// (unmapped bits default good). Without it the cached bOK is still
// FALSE on a fresh instance and Advance() gets rejected with
// REJECTED_PERMISSIVE_NOT_MET.
fb();
fb.Advance(eRequester := TcForge.E_Requester.PROG);
fb();
AssertEquals_DINT(
    Expected := TcForge.E_TwoPosActuator_State.Advancing,
    Actual   := fb.sts.state,
    Message  := 'Precondition: must be in Advancing');

fb.inAdvanced := TRUE;
fb();

AssertEquals_DINT(
    Expected := TcForge.E_TwoPosActuator_State.Advanced,
    Actual   := fb.sts.state,
    Message  := 'Advancing must complete to Advanced when inFbkAdvanced asserts');
AssertFalse(
    Condition := fb.sts.moving,
    Message   := 'moving must clear once the motion completes');

TEST_FINISHED();
END_METHOD

METHOD AdvancingFaultsOnBothFeedback
VAR
    fb : TcForge.FB_TwoPosActuator;
END_VAR
TEST('AdvancingFaultsOnBothFeedback');

// Warmup cycle so advancePermissives reports bOK before Advance().
fb();
fb.Advance(eRequester := TcForge.E_Requester.PROG);
fb();

// Simulate a stuck or failed retracted end-stop latching HIGH while the
// actuator is already reporting Advanced — classic dual-sensor fault.
fb.inAdvanced := TRUE;
fb.inRetracted := TRUE;
fb();

AssertEquals_DINT(
    Expected := TcForge.E_TwoPosActuator_State.Fault,
    Actual   := fb.sts.state,
    Message  := 'Both feedbacks while Advancing must trip to Fault');
AssertEquals_DINT(
    Expected := TcForge.E_TwoPosActuator_Fault.BothFeedbackOn,
    Actual   := fb.sts.header.faultCode,
    Message  := 'Fault code must be BothFeedbackOn — the highest-priority feedback fault');

TEST_FINISHED();
END_METHOD

METHOD AdvancedFaultsOnLostFeedback
VAR
    fb : TcForge.FB_TwoPosActuator;
END_VAR
TEST('AdvancedFaultsOnLostFeedback');

fb.inAdvanced := TRUE;
fb();
AssertEquals_DINT(
    Expected := TcForge.E_TwoPosActuator_State.Advanced,
    Actual   := fb.sts.state,
    Message  := 'Precondition: must be in Advanced');

// Feedback drops while the actuator is supposed to be at the end-stop
// (wire break, loose sensor, etc.). The FB must not silently revert to
// Undefined — that would let downstream sequencing assume a known state
// that isn't actually valid.
fb.inAdvanced := FALSE;
fb();

AssertEquals_DINT(
    Expected := TcForge.E_TwoPosActuator_State.Fault,
    Actual   := fb.sts.state,
    Message  := 'Lost advanced feedback must trip to Fault, not silently revert');
AssertEquals_DINT(
    Expected := TcForge.E_TwoPosActuator_Fault.UndefinedState,
    Actual   := fb.sts.header.faultCode,
    Message  := 'Fault code must be UndefinedState when Advanced feedback disappears');

TEST_FINISHED();
END_METHOD

METHOD RetractFromAdvancedDrivesRetracting
VAR
    fb   : TcForge.FB_TwoPosActuator;
    resp : TcForge.E_RpcMethodResponse;
END_VAR
TEST('RetractFromAdvancedDrivesRetracting');

fb.inAdvanced := TRUE;
fb();
fb.inAdvanced := FALSE;

resp := fb.Retract(eRequester := TcForge.E_Requester.PROG);
fb();

AssertEquals_DINT(
    Expected := TcForge.E_RpcMethodResponse.ACCEPTED,
    Actual   := resp,
    Message  := 'Retract from Advanced must be ACCEPTED');
AssertEquals_DINT(
    Expected := TcForge.E_TwoPosActuator_State.Retracting,
    Actual   := fb.sts.state,
    Message  := 'Accepted Retract must transition to Retracting');
AssertTrue(
    Condition := fb.outRetract,
    Message   := 'Retracting must energize outValveRetract');
AssertFalse(
    Condition := fb.outAdvance,
    Message   := 'Retracting must NOT energize outValveAdvance');

TEST_FINISHED();
END_METHOD

METHOD AbortAlwaysAcceptedAndReturnsToUndefined
VAR
    fb   : TcForge.FB_TwoPosActuator;
    resp : TcForge.E_RpcMethodResponse;
END_VAR
TEST('AbortAlwaysAcceptedAndReturnsToUndefined');

// Set up a worst-case: source-locked AND in motion AND commanded by
// OPERATOR. Abort must still land. Warmup cycle first so
// advancePermissives reports bOK before Advance().
fb();
fb.LockSource(bLock := TRUE);
fb.Advance(eRequester := TcForge.E_Requester.PROG);
fb();
AssertEquals_DINT(
    Expected := TcForge.E_TwoPosActuator_State.Advancing,
    Actual   := fb.sts.state,
    Message  := 'Precondition: must be Advancing before Abort');

resp := fb.Abort(eRequester := TcForge.E_Requester.OPERATOR);
fb();

AssertEquals_DINT(
    Expected := TcForge.E_RpcMethodResponse.ACCEPTED,
    Actual   := resp,
    Message  := 'Abort must be accepted from OPERATOR even when source-locked (safety invariant)');
AssertEquals_DINT(
    Expected := TcForge.E_TwoPosActuator_State.Undefined,
    Actual   := fb.sts.state,
    Message  := 'Abort must return state to Undefined for re-evaluation');
AssertFalse(
    Condition := fb.outAdvance,
    Message   := 'Abort must de-energize outValveAdvance');
AssertFalse(
    Condition := fb.outRetract,
    Message   := 'Abort must de-energize outValveRetract');

TEST_FINISHED();
END_METHOD

METHOD ResetClearsFaultAndReturnsToUndefined
VAR
    fb   : TcForge.FB_TwoPosActuator;
    resp : TcForge.E_RpcMethodResponse;
END_VAR
TEST('ResetClearsFaultAndReturnsToUndefined');

// Trip to Fault via the both-feedbacks path.
fb.inAdvanced := TRUE;
fb.inRetracted := TRUE;
fb();
AssertTrue(
    Condition := fb.sts.header.faulted,
    Message   := 'Precondition: must be faulted before Reset');

// Drop the conflicting feedback so Reset can actually settle.
fb.inRetracted := FALSE;
fb.inAdvanced := FALSE;

resp := fb.Reset(eRequester := TcForge.E_Requester.OPERATOR);
fb();

AssertEquals_DINT(
    Expected := TcForge.E_RpcMethodResponse.ACCEPTED,
    Actual   := resp,
    Message  := 'Reset must always be accepted (safety invariant inherited from FB_DeviceBase)');
AssertFalse(
    Condition := fb.sts.header.faulted,
    Message   := 'Reset must clear the active fault');
AssertEquals_DINT(
    Expected := TcForge.E_TwoPosActuator_State.Undefined,
    Actual   := fb.sts.state,
    Message  := 'Reset must drop the state machine back to Undefined');
AssertTrue(
    Condition := fb.sts.header.lastFaultCode = TcForge.E_TwoPosActuator_Fault.BothFeedbackOn,
    Message   := 'Reset must preserve lastFaultCode for HMI post-mortem');

TEST_FINISHED();
END_METHOD

METHOD HeaderBusyMirrorsMovingState
VAR
    fb : TcForge.FB_TwoPosActuator;
END_VAR
TEST('HeaderBusyMirrorsMovingState');

// Warmup cycle so advancePermissives reports bOK before Advance().
fb();
fb.Advance(eRequester := TcForge.E_Requester.PROG);
fb();

AssertTrue(
    Condition := fb.sts.moving,
    Message   := 'Advancing must set moving');
AssertTrue(
    Condition := fb.sts.header.busy,
    Message   := 'header.busy must mirror moving so generic HMIs can show motion');
AssertFalse(
    Condition := fb.sts.header.ready,
    Message   := 'ready must be FALSE while the actuator is in motion');

TEST_FINISHED();
END_METHOD

END_FUNCTION_BLOCK

// ---- Tests/FB_AnalogInput_Test.TcPOU
// Tests exercise the public input/output and command contracts.
FUNCTION_BLOCK FB_AnalogInput_Test EXTENDS TcUnit.FB_TestSuite
VAR CONSTANT
    TOL : REAL := 1E-3;
END_VAR

InitialStatusPublishesDefaults();
LinearScalingMapsEndpointsAndMidpoint();
RawBypassSkipsClampAndScaling();
ClampLowReportsAndHoldsAtRawMin();
ClampHighReportsAndHoldsAtRawMax();
ClampPromotesGoodQualityToClamped();
ClampAsFaultRaisesClampLow();
ClampAsFaultRaisesClampHigh();
BadConfigRaisesFaultOnFirstScan();
BadQualityHoldsLastRawReading();
InputTypeRealReadsRealMemberOfUnion();
QualityTagPropagatesToStatus();

METHOD InitialStatusPublishesDefaults
VAR
    fb : TcForge.FB_AnalogInput;
END_VAR
TEST('InitialStatusPublishesDefaults');

// Default cfg: INT terminal, raw 0..32767 -> EU 0..100, no filter,
// clamp-as-fault disabled. The application must explicitly label the unit.
// With inRaw zero-initialised the first cycle reports a clean 0 and no fault.
fb(inpQuality := TcForge.E_IO_Quality.GOOD);

AssertTrue(
    Condition := fb.sts.unit = TcForge.E_Unit.UNSPECIFIED,
    Message   := 'An unconfigured channel must not claim a physical unit');

AssertTrue(
    Condition := ABS(fb.sts.value) < TOL,
    Message   := 'Fresh instance must publish value = 0 for a raw input of 0');
AssertTrue(
    Condition := ABS(fb.sts.rawReal) < TOL,
    Message   := 'Fresh instance must publish rawReal = 0');
AssertFalse(
    Condition := fb.sts.clampActive,
    Message   := 'Raw 0 is inside [0, 32767] so clampActive must be FALSE');
AssertFalse(
    Condition := fb.sts.header.faulted,
    Message   := 'Fresh instance must not be faulted');

TEST_FINISHED();
END_METHOD

METHOD LinearScalingMapsEndpointsAndMidpoint
VAR
    fb : TcForge.FB_AnalogInput;
END_VAR
TEST('LinearScalingMapsEndpointsAndMidpoint');

// Default cfg: raw 0..32767 -> EU 0..100. Verify the two endpoints and
// the midpoint land where the linear recurrence says they should.
//
//     value = euMin + (raw - rawMin)
//                           * (euMax - euMin)
//                           / (rawMax - rawMin)

fb.inRaw.nInt := 0;
fb(inpQuality := TcForge.E_IO_Quality.GOOD);
AssertTrue(
    Condition := ABS(fb.sts.value - 0.0) < TOL,
    Message   := 'Raw = rawMin must map to euMin (0 %)');

fb.inRaw.nInt := 32767;
fb(inpQuality := TcForge.E_IO_Quality.GOOD);
AssertTrue(
    Condition := ABS(fb.sts.value - 100.0) < TOL,
    Message   := 'Raw = rawMax must map to euMax (100 %)');

fb.inRaw.nInt := 16384;
fb(inpQuality := TcForge.E_IO_Quality.GOOD);
AssertTrue(
    Condition := ABS(fb.sts.value - 50.0015) < 0.01,
    Message   := 'Raw ~ midpoint must map to EU ~ 50 %');

TEST_FINISHED();
END_METHOD

METHOD RawBypassSkipsClampAndScaling
VAR
    fb : TcForge.FB_AnalogInput;
END_VAR
TEST('RawBypassSkipsClampAndScaling');

// useRawValue = TRUE publishes the raw REAL directly and suppresses
// the clamp flags even when the raw value is outside the scaling range.
fb.cfg.useRawValue := TRUE;
fb.inRaw.nInt := 30000;
fb(inpQuality := TcForge.E_IO_Quality.GOOD);

AssertTrue(
    Condition := ABS(fb.sts.value - fb.sts.rawReal) < TOL,
    Message   := 'With useRawValue = TRUE, value must equal rawReal');
AssertFalse(
    Condition := fb.sts.clampedLow,
    Message   := 'Raw bypass must not flag clampedLow');
AssertFalse(
    Condition := fb.sts.clampedHigh,
    Message   := 'Raw bypass must not flag clampedHigh');
AssertFalse(
    Condition := fb.sts.clampActive,
    Message   := 'Raw bypass must not flag clampActive');

TEST_FINISHED();
END_METHOD

METHOD ClampLowReportsAndHoldsAtRawMin
VAR
    fb : TcForge.FB_AnalogInput;
END_VAR
TEST('ClampLowReportsAndHoldsAtRawMin');

// Drive the raw INT below rawMin. The clamp must flag clampedLow
// and pin the scaled value at euMin.
fb.inRaw.nInt := -500;
fb(inpQuality := TcForge.E_IO_Quality.GOOD);

AssertTrue(
    Condition := fb.sts.clampedLow,
    Message   := 'Raw below rawMin must set clampedLow');
AssertTrue(
    Condition := fb.sts.clampActive,
    Message   := 'clampActive must be TRUE whenever either clamp direction is active');
AssertTrue(
    Condition := ABS(fb.sts.value - 0.0) < TOL,
    Message   := 'Clamped-low output must pin to euMin (0 %)');
AssertFalse(
    Condition := fb.sts.header.faulted,
    Message   := 'clampAsFault = FALSE by default; clamp alone must not fault the device');

TEST_FINISHED();
END_METHOD

METHOD ClampHighReportsAndHoldsAtRawMax
VAR
    fb : TcForge.FB_AnalogInput;
END_VAR
TEST('ClampHighReportsAndHoldsAtRawMax');

// Use REAL input so we can inject a raw that is clearly above rawMax
// (INT saturates at 32767; REAL doesn't).
fb.cfg.inputType := __SYSTEM.TYPE_CLASS.TYPE_REAL;
fb.inRaw.fReal := 40000.0;
fb(inpQuality := TcForge.E_IO_Quality.GOOD);

